KUKA KRL program: MyProgram_149().src

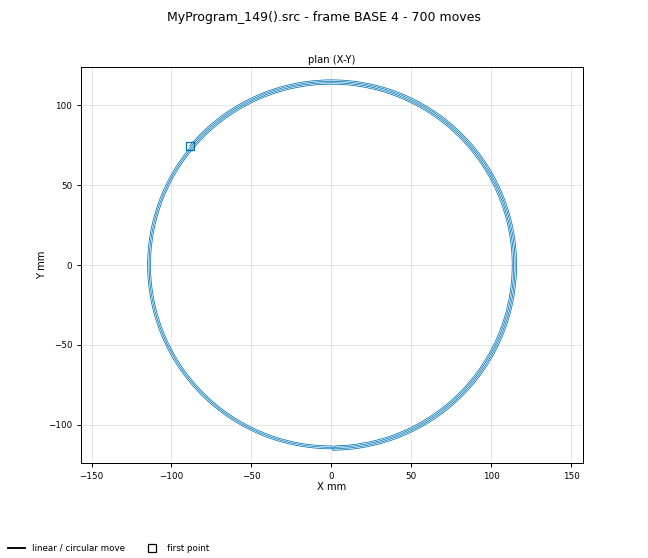
[picture p0: tool path of MyProgram_149().src in frame BASE 4, 700 of 700 moves have a stored position in this frame; points joined in program order, loops and branches not executed]
&ACCESS RVP
&REL 1
&PARAM TEMPLATE = C:\KRC\Roboter\Template\vorgabe
&PARAM EDITMASK = *
DEF MyProgram_149()
; ---- Setting reference (Base) ----
$BASE = BASE_DATA[4]

; --------------------------
; ---- Setting tool (TCP) ----
$TOOL = TOOL_DATA[3]
; --------------------------

$VEL.CP = VEL_APROX_PRINT
Startdeposition()
$VEL.CP = VEL_PRINT
LIN {X -88.6601,Y 74.5291,Z 117,A 135.3963,B 24.9406,C -1.7805,E1 24.8781,E2 310.5914} C_DIS
LIN {X -86.8043,Y 76.6825,Z 117,A 133.9686,B 24.9404,C -1.7832,E1 24.8807,E2 312.019} C_DIS
LIN {X -84.8592,Y 78.8302,Z 117,A 132.5273,B 24.9402,C -1.7865,E1 24.8834,E2 313.4588} C_DIS
LIN {X -82.9372,Y 80.8494,Z 117,A 131.1408,B 24.94,C -1.7896,E1 24.8861,E2 314.8439} C_DIS
LIN {X -80.928,Y 82.8605,Z 117,A 129.7272,B 24.9398,C -1.7928,E1 24.8889,E2 316.256} C_DIS
LIN {X -78.8302,Y 84.8592,Z 117,A 128.2864,B 24.9396,C -1.7958,E1 24.8918,E2 317.6954} C_DIS
LIN {X -77.0268,Y 86.497,Z 117,A 127.0345,B 24.9395,C -1.7968,E1 24.8944,E2 318.9501} C_DIS
LIN {X -74.5714,Y 88.625,Z 117,A 125.4601,B 24.9392,C -1.8017,E1 24.8978,E2 320.5189} C_DIS
LIN {X -72.3739,Y 90.4284,Z 117,A 124.0473,B 24.939,C -1.8045,E1 24.9008,E2 321.9303} C_DIS
LIN {X -70.1764,Y 92.1438,Z 117,A 122.6615,B 24.9388,C -1.8072,E1 24.9039,E2 323.3147} C_DIS
LIN {X -67.9234,Y 93.8167,Z 117,A 121.2662,B 24.9386,C -1.8098,E1 24.907,E2 324.7087} C_DIS
LIN {X -65.5706,Y 95.4762,Z 117,A 119.8357,B 24.9384,C -1.8124,E1 24.9103,E2 326.138} C_DIS
LIN {X -63.2077,Y 97.0566,Z 117,A 118.4237,B 24.9383,C -1.8149,E1 24.9136,E2 327.5486} C_DIS
LIN {X -60.7603,Y 98.6077,Z 117,A 116.9852,B 24.9381,C -1.8174,E1 24.917,E2 328.9857} C_DIS
LIN {X -58.3693,Y 100.0412,Z 117,A 115.6133,B 24.9379,C -1.8202,E1 24.9203,E2 330.3551} C_DIS
LIN {X -55.8486,Y 101.4702,Z 117,A 114.162,B 24.9378,C -1.822,E1 24.9238,E2 331.8064} C_DIS
LIN {X -53.3902,Y 102.7847,Z 117,A 112.7778,B 24.9376,C -1.8241,E1 24.9272,E2 333.1894} C_DIS
LIN {X -50.8516,Y 104.064,Z 117,A 111.3658,B 24.9375,C -1.8262,E1 24.9308,E2 334.6002} C_DIS
LIN {X -48.2327,Y 105.3038,Z 117,A 109.9286,B 24.9373,C -1.8282,E1 24.9344,E2 336.0362} C_DIS
LIN {X -45.6339,Y 106.4558,Z 117,A 108.5177,B 24.9373,C -1.8301,E1 24.938,E2 337.4458} C_DIS
LIN {X -43.0076,Y 107.5436,Z 117,A 107.1073,B 24.9371,C -1.8319,E1 24.9417,E2 338.8551} C_DIS
LIN {X -40.3554,Y 108.5667,Z 117,A 105.697,B 24.937,C -1.8336,E1 24.9453,E2 340.2643} C_DIS
LIN {X -37.6788,Y 109.5243,Z 117,A 104.2869,B 24.9369,C -1.8352,E1 24.949,E2 341.6734} C_DIS
LIN {X -34.9796,Y 110.416,Z 117,A 102.8769,B 24.9368,C -1.8368,E1 24.9528,E2 343.0823} C_DIS
LIN {X -32.312,Y 111.2256,Z 117,A 101.4947,B 24.9367,C -1.8382,E1 24.9565,E2 344.4636} C_DIS
LIN {X -29.5726,Y 111.9851,Z 117,A 100.0842,B 24.9366,C -1.8394,E1 24.9603,E2 345.8732} C_DIS
LIN {X -26.8155,Y 112.6771,Z 117,A 98.6751,B 24.9365,C -1.8407,E1 24.9641,E2 347.2813} C_DIS
LIN {X -24.0422,Y 113.3013,Z 117,A 97.2672,B 24.9365,C -1.8418,E1 24.9679,E2 348.6881} C_DIS
LIN {X -21.5271,Y 113.8047,Z 117,A 95.9717,B 24.9365,C -1.8418,E1 24.9715,E2 349.9852} C_DIS
LIN {X -18.8927,Y 114.2711,Z 117,A 94.6168,B 24.9365,C -1.8414,E1 24.9752,E2 351.3423} C_DIS
LIN {X -15.5877,Y 114.7706,Z 117,A 93.0146,B 24.9362,C -1.8446,E1 24.9796,E2 352.9381} C_DIS
LIN {X -12.8209,Y 115.1122,Z 117,A 91.6457,B 24.9362,C -1.8459,E1 24.9834,E2 354.305} C_DIS
LIN {X -9.9921,Y 115.3922,Z 117,A 90.226,B 24.9362,C -1.8459,E1 24.9874,E2 355.7252} C_DIS
LIN {X -7.1024,Y 115.6064,Z 117,A 88.7913,B 24.9361,C -1.8465,E1 24.9914,E2 357.1591} C_DIS
LIN {X -4.3917,Y 115.7403,Z 117,A 87.4449,B 24.9361,C -1.8468,E1 24.9951,E2 358.5052} C_DIS
LIN {X -1.4213,Y 115.8156,Z 117,A 85.9771,B 24.9361,C -1.8473,E1 24.9992,E2 359.972} C_DIS
LIN {X 1.4213,Y 115.8156,Z 117,A 84.5704,B 24.9361,C -1.8475,E1 25.0032,E2 361.378} C_DIS
LIN {X 4.2632,Y 115.7459,Z 117,A 83.1636,B 24.9361,C -1.8476,E1 25.0071,E2 362.7843} C_DIS
LIN {X 7.0476,Y 115.6094,Z 117,A 81.7846,B 24.9361,C -1.8476,E1 25.0109,E2 364.1626} C_DIS
LIN {X 9.9374,Y 115.3973,Z 117,A 80.3512,B 24.9361,C -1.8476,E1 25.0149,E2 365.5955} C_DIS
LIN {X 12.2215,Y 115.1757,Z 117,A 79.1531,B 24.9362,C -1.8447,E1 25.0183,E2 366.7997} C_DIS
LIN {X 15.5877,Y 114.7706,Z 117,A 77.54,B 24.936,C -1.8471,E1 25.0227,E2 368.4058} C_DIS
LIN {X 17.9447,Y 114.4239,Z 117,A 76.3162,B 24.9362,C -1.8448,E1 25.0261,E2 369.6339} C_DIS
LIN {X 20.7205,Y 113.9539,Z 117,A 74.924,B 24.9362,C -1.8443,E1 25.0299,E2 371.0257} C_DIS
LIN {X 23.9885,Y 113.313,Z 117,A 73.3247,B 24.9362,C -1.8456,E1 25.0343,E2 372.62} C_DIS
LIN {X 26.7087,Y 112.7025,Z 117,A 71.9472,B 24.9362,C -1.845,E1 25.038,E2 373.9971} C_DIS
LIN {X 29.4665,Y 112.0131,Z 117,A 70.5426,B 24.9362,C -1.8442,E1 25.0418,E2 375.4014} C_DIS
LIN {X 32.2594,Y 111.2412,Z 117,A 69.1115,B 24.9363,C -1.8433,E1 25.0457,E2 376.8323} C_DIS
LIN {X 34.9272,Y 110.4323,Z 117,A 67.7347,B 24.9363,C -1.8423,E1 25.0493,E2 378.2089} C_DIS
LIN {X 37.3427,Y 109.6377,Z 117,A 66.4515,B 24.9365,C -1.8401,E1 25.0528,E2 379.4947} C_DIS
LIN {X 40.3038,Y 108.5855,Z 117,A 64.9276,B 24.9365,C -1.8401,E1 25.0567,E2 381.0157} C_DIS
LIN {X 43.0076,Y 107.5436,Z 117,A 63.4973,B 24.9366,C -1.8387,E1 25.0605,E2 382.4459} C_DIS
LIN {X 45.4321,Y 106.5408,Z 117,A 62.1891,B 24.9368,C -1.8369,E1 25.0638,E2 383.7554} C_DIS
LIN {X 47.998,Y 105.4096,Z 117,A 60.8009,B 24.9368,C -1.8353,E1 25.0674,E2 385.144} C_DIS
LIN {X 50.8024,Y 104.0884,Z 117,A 59.2892,B 24.9369,C -1.8343,E1 25.0712,E2 386.654} C_DIS
LIN {X 53.2927,Y 102.8353,Z 117,A 57.9128,B 24.937,C -1.8327,E1 25.0746,E2 388.0306} C_DIS
LIN {X 55.8486,Y 101.4702,Z 117,A 56.4846,B 24.9372,C -1.8309,E1 25.0781,E2 389.4588} C_DIS
LIN {X 58.322,Y 100.0691,Z 117,A 55.0826,B 24.9372,C -1.8291,E1 25.0815,E2 390.8609} C_DIS
LIN {X 60.7133,Y 98.6362,Z 117,A 53.7195,B 24.9374,C -1.8277,E1 25.0848,E2 392.223} C_DIS
LIN {X 63.1157,Y 97.1165,Z 117,A 52.3067,B 24.9376,C -1.8252,E1 25.0881,E2 393.6373} C_DIS
LIN {X 65.1708,Y 95.7477,Z 117,A 51.045,B 24.9378,C -1.8214,E1 25.091,E2 394.9036} C_DIS
LIN {X 67.8497,Y 93.8707,Z 117,A 49.4771,B 24.9378,C -1.8208,E1 25.0946,E2 396.4674} C_DIS
LIN {X 70.089,Y 92.2103,Z 117,A 48.1024,B 24.938,C -1.8186,E1 25.0976,E2 397.8425} C_DIS
LIN {X 72.3739,Y 90.4284,Z 117,A 46.6755,B 24.9382,C -1.8162,E1 25.1008,E2 399.2697} C_DIS
LIN {X 75.2543,Y 88.0431,Z 117,A 44.7753,B 24.9386,C -1.8104,E1 25.1049,E2 401.1763} C_DIS
LIN {X 77.7829,Y 85.8202,Z 117,A 43.1751,B 24.9386,C -1.8099,E1 25.1082,E2 402.7712} C_DIS
LIN {X 79.8656,Y 83.8854,Z 117,A 41.7751,B 24.9388,C -1.8073,E1 25.111,E2 404.1717} C_DIS
LIN {X 81.9002,Y 81.9002,Z 117,A 40.3751,B 24.939,C -1.8046,E1 25.1138,E2 405.5723} C_DIS
LIN {X 83.8854,Y 79.8656,Z 117,A 38.9755,B 24.9392,C -1.8018,E1 25.1165,E2 406.9723} C_DIS
LIN {X 85.7831,Y 77.8233,Z 117,A 37.6053,B 24.9393,C -1.7991,E1 25.1191,E2 408.343} C_DIS
LIN {X 87.3549,Y 76.0521,Z 117,A 36.3734,B 24.9397,C -1.7936,E1 25.1214,E2 409.5821} C_DIS
LIN {X 89.5334,Y 73.4782,Z 117,A 34.778,B 24.9397,C -1.793,E1 25.1242,E2 411.1718} C_DIS
LIN {X 91.3097,Y 71.2588,Z 117,A 33.3787,B 24.94,C -1.7899,E1 25.1267,E2 412.5718} C_DIS
LIN {X 92.7838,Y 69.3256,Z 117,A 32.141,B 24.9403,C -1.7853,E1 25.1288,E2 413.8144} C_DIS
LIN {X 94.6962,Y 66.6926,Z 117,A 30.5813,B 24.9403,C -1.7835,E1 25.1313,E2 415.3707} C_DIS
LIN {X 96.3044,Y 64.3486,Z 117,A 29.1828,B 24.9406,C -1.7803,E1 25.1335,E2 416.77} C_DIS
LIN {X 97.7753,Y 62.0892,Z 117,A 27.8528,B 24.9408,C -1.7769,E1 25.1355,E2 418.1011} C_DIS
LIN {X 99.3459,Y 59.5456,Z 117,A 26.3861,B 24.941,C -1.7735,E1 25.1376,E2 419.5684} C_DIS
LIN {X 100.7561,Y 57.1265,Z 117,A 25.0092,B 24.9413,C -1.7702,E1 25.1395,E2 420.9462} C_DIS
LIN {X 102.1218,Y 54.6475,Z 117,A 23.6172,B 24.9415,C -1.7667,E1 25.1414,E2 422.3391} C_DIS
LIN {X 103.4321,Y 52.1248,Z 117,A 22.2197,B 24.9417,C -1.7631,E1 25.1432,E2 423.7375} C_DIS
LIN {X 104.704,Y 49.5213,Z 117,A 20.7949,B 24.942,C -1.7595,E1 25.1449,E2 425.1633} C_DIS
LIN {X 105.8877,Y 46.9368,Z 117,A 19.3972,B 24.9422,C -1.7558,E1 25.1465,E2 426.5621} C_DIS
LIN {X 107.0077,Y 44.3241,Z 117,A 17.9997,B 24.9425,C -1.7521,E1 25.148,E2 427.9607} C_DIS
LIN {X 108.0633,Y 41.6846,Z 117,A 16.6022,B 24.9427,C -1.7484,E1 25.1495,E2 429.3592} C_DIS
LIN {X 108.9986,Y 39.1713,Z 117,A 15.2768,B 24.943,C -1.7445,E1 25.1507,E2 430.6864} C_DIS
LIN {X 109.9785,Y 36.332,Z 117,A 13.8078,B 24.9432,C -1.7408,E1 25.152,E2 432.1558} C_DIS
LIN {X 110.837,Y 33.622,Z 117,A 12.4107,B 24.9435,C -1.7369,E1 25.1532,E2 433.5541} C_DIS
LIN {X 111.6138,Y 30.9446,Z 117,A 11.0407,B 24.9437,C -1.7331,E1 25.1542,E2 434.9252} C_DIS
LIN {X 112.2551,Y 28.5247,Z 117,A 9.7764,B 24.944,C -1.7281,E1 25.1551,E2 436.194} C_DIS
LIN {X 112.9058,Y 25.8284,Z 117,A 8.3965,B 24.9443,C -1.7234,E1 25.156,E2 437.5769} C_DIS
LIN {X 113.5878,Y 22.65,Z 117,A 6.8501,B 24.9445,C -1.7212,E1 25.1569,E2 439.1195} C_DIS
LIN {X 114.1094,Y 19.8556,Z 117,A 5.4522,B 24.9447,C -1.7172,E1 25.1576,E2 440.5188} C_DIS
LIN {X 114.5623,Y 17.0492,Z 117,A 4.0634,B 24.945,C -1.7135,E1 25.1582,E2 441.9081} C_DIS
LIN {X 114.9462,Y 14.2326,Z 117,A 2.6599,B 24.9453,C -1.7091,E1 25.1587,E2 443.3136} C_DIS
LIN {X 115.2666,Y 11.3528,Z 117,A 1.2365,B 24.9455,C -1.705,E1 25.1591,E2 444.7383} C_DIS
LIN {X 115.5061,Y 8.5753,Z 117,A -0.1344,B 24.9458,C -1.7009,E1 25.1594,E2 446.1106} C_DIS
LIN {X 115.6818,Y 5.738,Z 117,A -1.5297,B 24.946,C -1.6969,E1 25.1596,E2 447.5072} C_DIS
LIN {X 115.7878,Y 2.8973,Z 117,A -2.9272,B 24.9463,C -1.6927,E1 25.1598,E2 448.9062} C_DIS
LIN {X 115.8232,Y 0,Z 117,A -4.3066,B 24.9464,C -1.6906,E1 25.1598,E2 450.2824} C_DIS
LIN {X 115.7905,Y -2.7876,Z 117,A -5.7202,B 24.9468,C -1.6845,E1 25.1598,E2 451.7021} C_DIS
LIN {X 115.6848,Y -5.6832,Z 117,A -7.1426,B 24.9471,C -1.6803,E1 25.1595,E2 453.1257} C_DIS
LIN {X 115.5142,Y -8.4658,Z 117,A -8.5122,B 24.9473,C -1.6763,E1 25.1593,E2 454.4968} C_DIS
LIN {X 115.2666,Y -11.3528,Z 117,A -9.9355,B 24.9476,C -1.6721,E1 25.1589,E2 455.9216} C_DIS
LIN {X 115.0189,Y -13.6181,Z 117,A -11.1264,B 24.948,C -1.6654,E1 25.1585,E2 457.1211} C_DIS
LIN {X 114.5784,Y -16.9406,Z 117,A -12.7024,B 24.9481,C -1.6639,E1 25.1579,E2 458.6915} C_DIS
LIN {X 114.1282,Y -19.7474,Z 117,A -14.0981,B 24.9484,C -1.6598,E1 25.1573,E2 460.0886} C_DIS
LIN {X 113.6092,Y -22.5423,Z 117,A -15.4956,B 24.9486,C -1.6556,E1 25.1566,E2 461.4877} C_DIS
LIN {X 113.0101,Y -25.3773,Z 117,A -16.9181,B 24.9489,C -1.6515,E1 25.1557,E2 462.9116} C_DIS
LIN {X 112.423,Y -27.8569,Z 117,A -18.1889,B 24.9492,C -1.647,E1 25.1549,E2 464.1857} C_DIS
LIN {X 111.6287,Y -30.8918,Z 117,A -19.7114,B 24.9494,C -1.6434,E1 25.1538,E2 465.708} C_DIS
LIN {X 110.837,Y -33.622,Z 117,A -21.108,B 24.9496,C -1.6394,E1 25.1527,E2 467.106} C_DIS
LIN {X 109.9954,Y -36.2798,Z 117,A -22.4779,B 24.9499,C -1.6354,E1 25.1515,E2 468.4775} C_DIS
LIN {X 109.0719,Y -38.9682,Z 117,A -23.8756,B 24.9501,C -1.6314,E1 25.1502,E2 469.8769} C_DIS
LIN {X 108.1211,Y -41.5319,Z 117,A -25.2235,B 24.9504,C -1.6274,E1 25.1489,E2 471.2266} C_DIS
LIN {X 107.0284,Y -44.2732,Z 117,A -26.6685,B 24.9506,C -1.6236,E1 25.1473,E2 472.6727} C_DIS
LIN {X 105.9097,Y -46.8865,Z 117,A -28.0665,B 24.9508,C -1.6196,E1 25.1458,E2 474.0724} C_DIS
LIN {X 104.8874,Y -49.1273,Z 117,A -29.3169,B 24.9512,C -1.6144,E1 25.1443,E2 475.3283} C_DIS
LIN {X 103.4571,Y -52.0759,Z 117,A -30.8867,B 24.9513,C -1.6119,E1 25.1424,E2 476.8956} C_DIS
LIN {X 102.1479,Y -54.5992,Z 117,A -32.2841,B 24.9515,C -1.6081,E1 25.1406,E2 478.2945} C_DIS
LIN {X 100.804,Y -57.0417,Z 117,A -33.6543,B 24.9518,C -1.6045,E1 25.1387,E2 479.6662} C_DIS
LIN {X 99.3738,Y -59.4984,Z 117,A -35.0515,B 24.952,C -1.6008,E1 25.1367,E2 481.0649} C_DIS
LIN {X 97.8837,Y -61.9192,Z 117,A -36.4495,B 24.9522,C -1.5971,E1 25.1346,E2 482.4645} C_DIS
LIN {X 96.3044,Y -64.3486,Z 117,A -37.8741,B 24.9524,C -1.5935,E1 25.1325,E2 483.8907} C_DIS
LIN {X 94.6962,Y -66.6926,Z 117,A -39.2719,B 24.9526,C -1.5899,E1 25.1302,E2 485.29} C_DIS
LIN {X 93.031,Y -68.9965,Z 117,A -40.6701,B 24.9528,C -1.5864,E1 25.1279,E2 486.6897} C_DIS
LIN {X 91.3097,Y -71.2588,Z 117,A -42.0682,B 24.9531,C -1.583,E1 25.1255,E2 488.0893} C_DIS
LIN {X 89.568,Y -73.4355,Z 117,A -43.4392,B 24.9532,C -1.5796,E1 25.1231,E2 489.4617} C_DIS
LIN {X 87.7388,Y -75.6115,Z 117,A -44.8377,B 24.9534,C -1.5763,E1 25.1206,E2 490.8617} C_DIS
LIN {X 85.8202,Y -77.7829,Z 117,A -46.2631,B 24.9536,C -1.573,E1 25.1179,E2 492.2887} C_DIS
LIN {X 83.8854,Y -79.8656,Z 117,A -47.6618,B 24.9538,C -1.5698,E1 25.1153,E2 493.6888} C_DIS
LIN {X 81.9002,Y -81.9002,Z 117,A -49.0605,B 24.954,C -1.5666,E1 25.1125,E2 495.089} C_DIS
LIN {X 79.9051,Y -83.8473,Z 117,A -50.4328,B 24.9542,C -1.5636,E1 25.1097,E2 496.4627} C_DIS
LIN {X 77.9197,Y -85.6946,Z 117,A -51.7743,B 24.9544,C -1.5604,E1 25.107,E2 497.8062} C_DIS
LIN {X 75.8953,Y -87.4919,Z 117,A -53.1262,B 24.9546,C -1.5567,E1 25.1041,E2 499.1615} C_DIS
LIN {X 73.5526,Y -89.4716,Z 117,A -54.6127,B 24.9547,C -1.5547,E1 25.101,E2 500.6471} C_DIS
LIN {X 71.3019,Y -91.2757,Z 117,A -56.03,B 24.9549,C -1.552,E1 25.0978,E2 502.0655} C_DIS
LIN {X 69.0404,Y -92.998,Z 117,A -57.43,B 24.955,C -1.5493,E1 25.0947,E2 503.4669} C_DIS
LIN {X 66.6926,Y -94.6962,Z 117,A -58.8567,B 24.9552,C -1.5466,E1 25.0915,E2 504.8949} C_DIS
LIN {X 64.3486,Y -96.3044,Z 117,A -60.2571,B 24.9553,C -1.544,E1 25.0882,E2 506.2966} C_DIS
LIN {X 61.966,Y -97.8545,Z 117,A -61.6573,B 24.9555,C -1.5416,E1 25.0849,E2 507.6982} C_DIS
LIN {X 59.5456,Y -99.3458,Z 117,A -63.0579,B 24.9556,C -1.5392,E1 25.0816,E2 509.1} C_DIS
LIN {X 57.0896,Y -100.7773,Z 117,A -64.4588,B 24.9557,C -1.5368,E1 25.0782,E2 510.5023} C_DIS
LIN {X 54.6475,Y -102.1218,Z 117,A -65.8328,B 24.9559,C -1.5347,E1 25.0748,E2 511.8774} C_DIS
LIN {X 52.1248,Y -103.4321,Z 117,A -67.2339,B 24.9559,C -1.5325,E1 25.0713,E2 513.2797} C_DIS
LIN {X 49.5213,Y -104.704,Z 117,A -68.6624,B 24.9561,C -1.5304,E1 25.0677,E2 514.7094} C_DIS
LIN {X 47.1001,Y -105.8142,Z 117,A -69.9814,B 24.9562,C -1.5283,E1 25.0644,E2 516.0301} C_DIS
LIN {X 44.3241,Y -107.0077,Z 117,A -71.4657,B 24.9563,C -1.5266,E1 25.0606,E2 517.5151} C_DIS
LIN {X 41.6846,Y -108.0633,Z 117,A -72.8677,B 24.9564,C -1.5248,E1 25.0569,E2 518.9182} C_DIS
LIN {X 39.0716,Y -109.0349,Z 117,A -74.2406,B 24.9565,C -1.5232,E1 25.0533,E2 520.2919} C_DIS
LIN {X 36.7201,Y -109.8476,Z 117,A -75.5113,B 24.9567,C -1.5199,E1 25.0499,E2 521.568} C_DIS
LIN {X 33.622,Y -110.837,Z 117,A -77.0751,B 24.9567,C -1.5199,E1 25.0458,E2 523.1288} C_DIS
LIN {X 30.9446,Y -111.6138,Z 117,A -78.4508,B 24.9567,C -1.5186,E1 25.0421,E2 524.5054} C_DIS
LIN {X 28.143,Y -112.3532,Z 117,A -79.8811,B 24.9569,C -1.5172,E1 25.0382,E2 525.9368} C_DIS
LIN {X 25.3773,Y -113.0101,Z 117,A -81.2845,B 24.9569,C -1.516,E1 25.0344,E2 527.3411} C_DIS
LIN {X 22.65,Y -113.5878,Z 117,A -82.6618,B 24.957,C -1.5149,E1 25.0306,E2 528.7194} C_DIS
LIN {X 19.8015,Y -114.1191,Z 117,A -84.092,B 24.957,C -1.5139,E1 25.0267,E2 530.1504} C_DIS
LIN {X 17.0492,Y -114.5623,Z 117,A -85.4699,B 24.9571,C -1.5129,E1 25.0229,E2 531.5292} C_DIS
LIN {X 14.2326,Y -114.9462,Z 117,A -86.8675,B 24.9571,C -1.5124,E1 25.019,E2 532.927} C_DIS
LIN {X 11.3528,Y -115.2666,Z 117,A -88.3045,B 24.9572,C -1.5114,E1 25.015,E2 534.3654} C_DIS
LIN {X 8.5206,Y -115.5105,Z 117,A -89.7097,B 24.9572,C -1.5107,E1 25.0111,E2 535.7713} C_DIS
LIN {X 5.6832,Y -115.6848,Z 117,A -91.1143,B 24.9572,C -1.5102,E1 25.0072,E2 537.1767} C_DIS
LIN {X 2.8973,Y -115.7878,Z 117,A -92.4935,B 24.9572,C -1.5098,E1 25.0033,E2 538.5567} C_DIS
LIN {X 0.8116,Y -115.8194,Z 117,A -93.2511,B 24.9566,C -1.5217,E1 25.0013,E2 539.2858} C_DIS
Enddeposition()
LIN {X 0.8116,Y -115.8194,Z 117,A -93.2511,B 24.9566,C -1.5217,E1 25.0013,E2 539.2858} C_DIS
Startdeposition()
$VEL.CP = VEL_PRINT
LIN {X 1.2098,Y -114.9149,Z 117,A -92.7013,B 24.9548,C -1.5531,E1 25.0031,E2 538.6618} C_DIS
LIN {X 3.6789,Y -114.8613,Z 117,A -91.2682,B 24.9543,C -1.5625,E1 25.0071,E2 537.2068} C_DIS
LIN {X 7.8843,Y -114.6494,Z 117,A -89.5393,B 24.9552,C -1.5468,E1 25.0118,E2 535.5156} C_DIS
LIN {X 11.3435,Y -114.3604,Z 117,A -87.5384,B 24.9544,C -1.5598,E1 25.0175,E2 533.4852} C_DIS
LIN {X 14.8457,Y -113.9572,Z 117,A -85.8672,B 24.9546,C -1.557,E1 25.0221,E2 531.8217} C_DIS
LIN {X 18.1047,Y -113.4864,Z 117,A -84.1715,B 24.9544,C -1.5606,E1 25.0268,E2 530.1191} C_DIS
LIN {X 20.9728,Y -112.992,Z 117,A -82.8451,B 24.9546,C -1.5562,E1 25.0304,E2 528.8047} C_DIS
LIN {X 25.3486,Y -112.0909,Z 117,A -80.5045,B 24.9542,C -1.5633,E1 25.0368,E2 526.4503} C_DIS
LIN {X 28.3498,Y -111.3687,Z 117,A -79.1593,B 24.9546,C -1.5561,E1 25.0404,E2 525.1241} C_DIS
LIN {X 30.6536,Y -110.7586,Z 117,A -77.8777,B 24.9543,C -1.5616,E1 25.0439,E2 523.8316} C_DIS
LIN {X 32.906,Y -110.1085,Z 117,A -76.5354,B 24.9538,C -1.5708,E1 25.0475,E2 522.4697} C_DIS
LIN {X 36.4786,Y -108.9771,Z 117,A -74.7175,B 24.9538,C -1.5708,E1 25.0524,E2 520.6553} C_DIS
LIN {X 40.4692,Y -107.559,Z 117,A -72.8108,B 24.9542,C -1.5643,E1 25.0573,E2 518.7679} C_DIS
LIN {X 42.6984,Y -106.6956,Z 117,A -71.3945,B 24.9535,C -1.5762,E1 25.0611,E2 517.3266} C_DIS
LIN {X 46.2055,Y -105.2225,Z 117,A -69.6792,B 24.9538,C -1.5708,E1 25.0654,E2 515.6283} C_DIS
LIN {X 49.1533,Y -103.88,Z 117,A -67.8577,B 24.9531,C -1.5828,E1 25.0701,E2 513.783} C_DIS
LIN {X 52.8895,Y -102.0283,Z 117,A -65.8043,B 24.9529,C -1.5851,E1 25.0752,E2 511.7298} C_DIS
LIN {X 56.3625,Y -100.1501,Z 117,A -63.4079,B 24.9515,C -1.6085,E1 25.0812,E2 509.2852} C_DIS
LIN {X 59.9119,Y -98.0677,Z 117,A -61.9666,B 24.953,C -1.584,E1 25.0845,E2 507.9062} C_DIS
LIN {X 61.8888,Y -96.8322,Z 117,A -60.7786,B 24.9528,C -1.5874,E1 25.0873,E2 506.7139} C_DIS
LIN {X 64.1436,Y -95.3538,Z 117,A -59.5511,B 24.9529,C -1.5847,E1 25.0901,E2 505.497} C_DIS
LIN {X 66.0888,Y -94.0174,Z 117,A -57.9839,B 24.9517,C -1.6052,E1 25.0938,E2 503.8867} C_DIS
LIN {X 69.9248,Y -91.1989,Z 117,A -55.8663,B 24.9521,C -1.5984,E1 25.0985,E2 501.7928} C_DIS
LIN {X 72.3813,Y -89.2613,Z 117,A -54.2134,B 24.9517,C -1.6062,E1 25.1021,E2 500.1276} C_DIS
LIN {X 75.2854,Y -86.8269,Z 117,A -52.645,B 24.9523,C -1.5956,E1 25.1053,E2 498.5904} C_DIS
LIN {X 77.4854,Y -84.8689,Z 117,A -50.9734,B 24.9515,C -1.6085,E1 25.1089,E2 496.8951} C_DIS
LIN {X 80.0003,Y -82.5028,Z 117,A -49.3117,B 24.9515,C -1.6099,E1 25.1122,E2 495.237} C_DIS
LIN {X 82.4878,Y -80.0159,Z 117,A -47.5085,B 24.951,C -1.6165,E1 25.1158,E2 493.4259} C_DIS
LIN {X 86.1776,Y -76.0289,Z 117,A -44.7625,B 24.9505,C -1.6252,E1 25.1209,E2 490.6715} C_DIS
LIN {X 88.1306,Y -73.7549,Z 117,A -43.2861,B 24.9503,C -1.6283,E1 25.1236,E2 489.1945} C_DIS
LIN {X 90.0442,Y -71.4053,Z 117,A -41.9968,B 24.9507,C -1.622,E1 25.1258,E2 487.9262} C_DIS
LIN {X 91.4747,Y -69.5663,Z 117,A -40.7691,B 24.9503,C -1.6282,E1 25.1279,E2 486.6896} C_DIS
LIN {X 92.8911,Y -67.6606,Z 117,A -39.5379,B 24.95,C -1.6337,E1 25.13,E2 485.4513} C_DIS
LIN {X 94.7831,Y -64.9865,Z 117,A -37.6998,B 24.9491,C -1.648,E1 25.1329,E2 483.5886} C_DIS
LIN {X 96.9625,Y -61.6857,Z 117,A -35.9075,B 24.9493,C -1.6451,E1 25.1356,E2 481.812} C_DIS
LIN {X 98.8733,Y -58.5723,Z 117,A -34.3784,B 24.9498,C -1.6367,E1 25.1378,E2 480.3107} C_DIS
LIN {X 100.2696,Y -56.1485,Z 117,A -32.9516,B 24.9495,C -1.6423,E1 25.1398,E2 478.878} C_DIS
LIN {X 101.2258,Y -54.4074,Z 117,A -31.4637,B 24.9478,C -1.6687,E1 25.1418,E2 477.3356} C_DIS
LIN {X 103.4745,Y -49.9973,Z 117,A -29.3447,B 24.9484,C -1.6596,E1 25.1444,E2 475.2493} C_DIS
LIN {X 105.0569,Y -46.5842,Z 117,A -27.5157,B 24.9482,C -1.6631,E1 25.1465,E2 473.422} C_DIS
LIN {X 105.9765,Y -44.4484,Z 117,A -26.1858,B 24.9474,C -1.6748,E1 25.148,E2 472.0719} C_DIS
LIN {X 107.2645,Y -41.2469,Z 117,A -24.4408,B 24.947,C -1.6813,E1 25.1498,E2 470.3213} C_DIS
LIN {X 108.3971,Y -38.167,Z 117,A -23.1047,B 24.9476,C -1.6722,E1 25.151,E2 469.014} C_DIS
LIN {X 109.1361,Y -36.0054,Z 117,A -21.9046,B 24.9472,C -1.6787,E1 25.1521,E2 467.8054} C_DIS
LIN {X 110.1267,Y -32.8448,Z 117,A -20.1785,B 24.9466,C -1.6875,E1 25.1535,E2 466.0684} C_DIS
LIN {X 110.935,Y -30.0011,Z 117,A -18.2953,B 24.9451,C -1.7117,E1 25.1549,E2 464.139} C_DIS
LIN {X 111.8375,Y -26.4452,Z 117,A -16.8441,B 24.9459,C -1.6996,E1 25.1558,E2 462.7248} C_DIS
LIN {X 112.5437,Y -23.2504,Z 117,A -15.2997,B 24.9458,C -1.7007,E1 25.1567,E2 461.1866} C_DIS
LIN {X 113.2613,Y -19.4624,Z 117,A -13.1544,B 24.9447,C -1.7176,E1 25.1578,E2 459.0143} C_DIS
LIN {X 113.9297,Y -15.0582,Z 117,A -11.1354,B 24.9449,C -1.7152,E1 25.1586,E2 457.0127} C_DIS
LIN {X 114.3995,Y -10.933,Z 117,A -9.0557,B 24.9444,C -1.7224,E1 25.1592,E2 454.9284} C_DIS
LIN {X 114.6916,Y -7.2602,Z 117,A -7.2779,B 24.9442,C -1.7256,E1 25.1595,E2 453.1535} C_DIS
LIN {X 114.8648,Y -3.5644,Z 117,A -5.4181,B 24.9438,C -1.7323,E1 25.1597,E2 451.2889} C_DIS
LIN {X 114.9209,Y 0.0447,Z 117,A -3.5719,B 24.9432,C -1.7404,E1 25.1597,E2 449.4346} C_DIS
LIN {X 114.8458,Y 4.1853,Z 117,A -1.4924,B 24.9427,C -1.7478,E1 25.1597,E2 447.3501} C_DIS
LIN {X 114.624,Y 8.2601,Z 117,A 0.4468,B 24.9427,C -1.7499,E1 25.1593,E2 445.4175} C_DIS
LIN {X 114.3962,Y 10.9685,Z 117,A 2.3157,B 24.9407,C -1.7787,E1 25.1588,E2 443.4919} C_DIS
LIN {X 113.9176,Y 15.1513,Z 117,A 3.9305,B 24.9418,C -1.7623,E1 25.1582,E2 441.9251} C_DIS
LIN {X 113.3315,Y 19.0424,Z 117,A 5.6967,B 24.942,C -1.7593,E1 25.1574,E2 440.1764} C_DIS
LIN {X 111.8917,Y 26.211,Z 117,A 9.4772,B 24.9408,C -1.7771,E1 25.1553,E2 436.376} C_DIS
LIN {X 110.9136,Y 30.0801,Z 117,A 11.2864,B 24.941,C -1.7747,E1 25.154,E2 434.5827} C_DIS
LIN {X 110.0384,Y 33.1422,Z 117,A 12.9677,B 24.9403,C -1.784,E1 25.1527,E2 432.8893} C_DIS
LIN {X 108.9126,Y 36.6699,Z 117,A 14.6469,B 24.9405,C -1.7817,E1 25.1512,E2 431.2248} C_DIS
LIN {X 108.1143,Y 38.9631,Z 117,A 15.8161,B 24.9404,C -1.7834,E1 25.1501,E2 430.0582} C_DIS
LIN {X 106.9404,Y 42.0761,Z 117,A 17.6294,B 24.9396,C -1.7956,E1 25.1483,E2 428.2263} C_DIS
LIN {X 105.5383,Y 45.4811,Z 117,A 19.3784,B 24.9395,C -1.7969,E1 25.1464,E2 426.484} C_DIS
LIN {X 104.2964,Y 48.2593,Z 117,A 21.1725,B 24.9383,C -1.8142,E1 25.1443,E2 424.6586} C_DIS
LIN {X 102.6069,Y 51.7574,Z 117,A 22.8621,B 24.9387,C -1.8081,E1 25.1422,E2 422.9926} C_DIS
LIN {X 101.1138,Y 54.6139,Z 117,A 24.3154,B 24.9389,C -1.8054,E1 25.1404,E2 421.5532} C_DIS
LIN {X 100.0352,Y 56.5683,Z 117,A 25.755,B 24.9377,C -1.8237,E1 25.1383,E2 420.0781} C_DIS
LIN {X 97.7913,Y 60.3646,Z 117,A 27.689,B 24.9381,C -1.8172,E1 25.1356,E2 418.1691} C_DIS
LIN {X 96.5777,Y 62.2852,Z 117,A 29.1257,B 24.9369,C -1.8344,E1 25.1334,E2 416.6992} C_DIS
LIN {X 94.3098,Y 65.6682,Z 117,A 30.989,B 24.9371,C -1.8318,E1 25.1305,E2 414.8512} C_DIS
LIN {X 92.1315,Y 68.692,Z 117,A 32.6995,B 24.9373,C -1.8296,E1 25.1277,E2 413.154} C_DIS
LIN {X 88.04,Y 73.8639,Z 117,A 36.1641,B 24.9361,C -1.8456,E1 25.1216,E2 409.6677} C_DIS
LIN {X 84.0193,Y 78.4066,Z 117,A 38.8882,B 24.9366,C -1.8387,E1 25.1165,E2 406.9722} C_DIS
LIN {X 81.8636,Y 80.6536,Z 117,A 40.5703,B 24.936,C -1.848,E1 25.1132,E2 405.2752} C_DIS
LIN {X 79.6601,Y 82.8307,Z 117,A 43.3096,B 24.9319,C -1.9066,E1 25.1075,E2 402.4088} C_DIS
LIN {X 74.5872,Y 87.4265,Z 117,A 45.8601,B 24.9342,C -1.8734,E1 25.1022,E2 399.9469} C_DIS
LIN {X 70.5238,Y 90.7373,Z 117,A 48.223,B 24.9347,C -1.8667,E1 25.0971,E2 397.6084} C_DIS
LIN {X 67.3246,Y 93.1371,Z 117,A 50.1355,B 24.9347,C -1.8665,E1 25.0928,E2 395.7033} C_DIS
LIN {X 64.5759,Y 95.0612,Z 117,A 51.86,B 24.9343,C -1.8717,E1 25.0889,E2 393.9723} C_DIS
LIN {X 61.1525,Y 97.2991,Z 117,A 53.6095,B 24.935,C -1.8619,E1 25.0848,E2 392.2519} C_DIS
LIN {X 58.5283,Y 98.8993,Z 117,A 55.1659,B 24.9348,C -1.8653,E1 25.0811,E2 390.6923} C_DIS
LIN {X 56.0201,Y 100.3413,Z 117,A 56.7599,B 24.9342,C -1.8742,E1 25.0772,E2 389.0821} C_DIS
LIN {X 53.1749,Y 101.8786,Z 117,A 58.2881,B 24.9342,C -1.8725,E1 25.0734,E2 387.562} C_DIS
LIN {X 46.1341,Y 105.2536,Z 117,A 62.1275,B 24.9342,C -1.8748,E1 25.0638,E2 383.7272} C_DIS
LIN {X 42.9658,Y 106.5867,Z 117,A 64.1238,B 24.9331,C -1.8892,E1 25.0585,E2 381.7014} C_DIS
LIN {X 39.5139,Y 107.9134,Z 117,A 65.8727,B 24.9333,C -1.8867,E1 25.054,E2 379.9621} C_DIS
LIN {X 35.6771,Y 109.2423,Z 117,A 67.8133,B 24.9334,C -1.8847,E1 25.0489,E2 378.03} C_DIS
LIN {X 32.0211,Y 110.371,Z 117,A 69.8116,B 24.933,C -1.8901,E1 25.0435,E2 376.0224} C_DIS
LIN {X 28.805,Y 111.2517,Z 117,A 71.472,B 24.933,C -1.8911,E1 25.039,E2 374.3623} C_DIS
LIN {X 24.1663,Y 112.3509,Z 117,A 73.7292,B 24.9332,C -1.8871,E1 25.0329,E2 372.1177} C_DIS
LIN {X 19.824,Y 113.1986,Z 117,A 76.1268,B 24.9326,C -1.8964,E1 25.0263,E2 369.7007} C_DIS
LIN {X 17.0102,Y 113.6556,Z 117,A 77.9714,B 24.9312,C -1.9155,E1 25.0211,E2 367.8128} C_DIS
LIN {X 12.9971,Y 114.1834,Z 117,A 79.3582,B 24.9332,C -1.8881,E1 25.0174,E2 366.4917} C_DIS
LIN {X 8.8009,Y 114.5832,Z 117,A 81.5091,B 24.933,C -1.8905,E1 25.0114,E2 364.3365} C_DIS
LIN {X 5.1762,Y 114.8037,Z 117,A 83.6805,B 24.9319,C -1.9061,E1 25.0053,E2 362.1287} C_DIS
LIN {X -0.609,Y 114.9185,Z 117,A 86.365,B 24.9325,C -1.8969,E1 24.9978,E2 359.4663} C_DIS
LIN {X -4.9468,Y 114.8136,Z 117,A 88.2754,B 24.9334,C -1.8854,E1 24.9926,E2 357.583} C_DIS
LIN {X -11.0074,Y 114.3926,Z 117,A 91.3713,B 24.9333,C -1.8868,E1 24.9839,E2 354.4823} C_DIS
LIN {X -16.4611,Y 113.7355,Z 117,A 94.3856,B 24.9325,C -1.897,E1 24.9755,E2 351.4418} C_DIS
LIN {X -23.3014,Y 112.5332,Z 117,A 97.7356,B 24.9331,C -1.8894,E1 24.9664,E2 348.1063} C_DIS
LIN {X -27.1679,Y 111.6626,Z 117,A 99.6627,B 24.9334,C -1.8855,E1 24.9611,E2 346.1859} C_DIS
LIN {X -29.8429,Y 110.9777,Z 117,A 101.151,B 24.9331,C -1.8888,E1 24.9571,E2 344.6874} C_DIS
LIN {X -33.1987,Y 110.0217,Z 117,A 102.8773,B 24.9333,C -1.8863,E1 24.9525,E2 342.9643} C_DIS
LIN {X -36.0859,Y 109.1095,Z 117,A 104.3798,B 24.9335,C -1.8841,E1 24.9485,E2 341.4641} C_DIS
LIN {X -38.9619,Y 108.1148,Z 117,A 105.8393,B 24.9338,C -1.8798,E1 24.9447,E2 340.012} C_DIS
LIN {X -42.4698,Y 106.7857,Z 117,A 107.5593,B 24.9344,C -1.8709,E1 24.9402,E2 338.3094} C_DIS
LIN {X -45.8461,Y 105.3792,Z 117,A 109.3994,B 24.9345,C -1.869,E1 24.9355,E2 336.4697} C_DIS
LIN {X -48.1855,Y 104.3308,Z 117,A 110.7297,B 24.9345,C -1.8692,E1 24.9321,E2 335.1356} C_DIS
LIN {X -52.8127,Y 102.0675,Z 117,A 114.0614,B 24.9325,C -1.8971,E1 24.9236,E2 331.7288} C_DIS
LIN {X -56.9846,Y 99.7973,Z 117,A 115.7506,B 24.9348,C -1.8644,E1 24.9197,E2 330.1122} C_DIS
LIN {X -60.6889,Y 97.5886,Z 117,A 117.6465,B 24.9359,C -1.8499,E1 24.9152,E2 328.2451} C_DIS
LIN {X -63.2677,Y 95.9366,Z 117,A 119.4564,B 24.9352,C -1.8587,E1 24.9109,E2 326.4085} C_DIS
LIN {X -66.5422,Y 93.6954,Z 117,A 121.1598,B 24.9363,C -1.8433,E1 24.9071,E2 324.7358} C_DIS
LIN {X -68.866,Y 92.0008,Z 117,A 122.7258,B 24.9361,C -1.8458,E1 24.9035,E2 323.1584} C_DIS
LIN {X -71.8267,Y 89.7108,Z 117,A 124.672,B 24.9361,C -1.845,E1 24.8993,E2 321.2069} C_DIS
LIN {X -74.5606,Y 87.4492,Z 117,A 126.5696,B 24.9361,C -1.8464,E1 24.8952,E2 319.2987} C_DIS
LIN {X -77.7773,Y 84.601,Z 117,A 128.7402,B 24.9364,C -1.8426,E1 24.8907,E2 317.1285} C_DIS
LIN {X -80.3588,Y 82.1548,Z 117,A 130.4178,B 24.9369,C -1.8344,E1 24.8873,E2 315.4635} C_DIS
LIN {X -82.1903,Y 80.3229,Z 117,A 131.878,B 24.9367,C -1.8381,E1 24.8844,E2 313.9882} C_DIS
LIN {X -85.0516,Y 77.2863,Z 117,A 133.9655,B 24.937,C -1.8331,E1 24.8805,E2 311.9032} C_DIS
LIN {X -87.1459,Y 74.9166,Z 117,A 135.4008,B 24.9377,C -1.8233,E1 24.8779,E2 310.4849} C_DIS
LIN {X -89.7971,Y 71.7179,Z 117,A 137.571,B 24.9377,C -1.8218,E1 24.8741,E2 308.308} C_DIS
LIN {X -92.26,Y 68.5209,Z 117,A 139.4837,B 24.9384,C -1.8123,E1 24.8708,E2 306.4088} C_DIS
LIN {X -94.1347,Y 65.9201,Z 117,A 141.2197,B 24.9384,C -1.8135,E1 24.868,E2 304.6615} C_DIS
LIN {X -95.6699,Y 63.6722,Z 117,A 143.0397,B 24.9373,C -1.8286,E1 24.8652,E2 302.7966} C_DIS
LIN {X -97.8841,Y 60.214,Z 117,A 144.6181,B 24.939,C -1.8036,E1 24.8629,E2 301.2697} C_DIS
LIN {X -99.9434,Y 56.7303,Z 117,A 146.7418,B 24.9391,C -1.802,E1 24.8599,E2 299.1387} C_DIS
LIN {X -101.7013,Y 53.5115,Z 117,A 148.4792,B 24.9397,C -1.7929,E1 24.8577,E2 297.4138} C_DIS
LIN {X -103.2186,Y 50.5261,Z 117,A 150.2626,B 24.9397,C -1.7925,E1 24.8554,E2 295.6218} C_DIS
LIN {X -105.3423,Y 45.9307,Z 117,A 152.8863,B 24.94,C -1.7889,E1 24.8524,E2 292.9923} C_DIS
LIN {X -107.0883,Y 41.6996,Z 117,A 154.7958,B 24.9415,C -1.7668,E1 24.8505,E2 291.1249} C_DIS
LIN {X -108.4159,Y 38.1134,Z 117,A 156.8745,B 24.9415,C -1.7677,E1 24.8485,E2 289.032} C_DIS
LIN {X -109.3777,Y 35.2586,Z 117,A 158.2675,B 24.942,C -1.7586,E1 24.8473,E2 287.6529} C_DIS
LIN {X -110.0718,Y 33.0297,Z 117,A 159.5635,B 24.942,C -1.7602,E1 24.8462,E2 286.3455} C_DIS
LIN {X -111.0529,Y 29.5646,Z 117,A 161.2652,B 24.9426,C -1.7507,E1 24.845,E2 284.6566} C_DIS
LIN {X -111.6296,Y 27.3032,Z 117,A 162.4051,B 24.9429,C -1.7461,E1 24.8442,E2 283.5211} C_DIS
LIN {X -112.3368,Y 24.2312,Z 117,A 164.1946,B 24.9426,C -1.7498,E1 24.8431,E2 281.7123} C_DIS
LIN {X -113.0969,Y 20.3896,Z 117,A 165.9097,B 24.9437,C -1.7339,E1 24.8422,E2 280.0248} C_DIS
LIN {X -113.523,Y 17.8679,Z 117,A 167.2351,B 24.9437,C -1.7318,E1 24.8416,E2 278.6966} C_DIS
LIN {X -113.9003,Y 15.2852,Z 117,A 168.5271,B 24.9441,C -1.7272,E1 24.8411,E2 277.4079} C_DIS
LIN {X -114.1881,Y 12.9572,Z 117,A 169.9757,B 24.9436,C -1.7346,E1 24.8406,E2 275.9329} C_DIS
LIN {X -114.5756,Y 8.8964,Z 117,A 171.9711,B 24.9441,C -1.7265,E1 24.8402,E2 273.945} C_DIS
LIN {X -114.743,Y 6.3783,Z 117,A 173.6692,B 24.9432,C -1.7402,E1 24.8399,E2 272.2039} C_DIS
LIN {X -114.8944,Y 2.4552,Z 117,A 175.5738,B 24.9438,C -1.7317,E1 24.8398,E2 270.3082} C_DIS
LIN {X -114.915,Y -1.1737,Z 117,A 177.0643,B 24.945,C -1.7129,E1 24.8398,E2 268.8535} C_DIS
LIN {X -114.6943,Y -7.2201,Z 117,A -179.939,B 24.9457,C -1.7023,E1 24.8402,E2 265.864} C_DIS
LIN {X -114.395,Y -10.9812,Z 117,A -177.9865,B 24.9459,C -1.6991,E1 24.8407,E2 263.9074} C_DIS
LIN {X -113.9345,Y -15.0207,Z 117,A -176.0827,B 24.9466,C -1.6877,E1 24.8413,E2 262.0195} C_DIS
LIN {X -113.4172,Y -18.5297,Z 117,A -174.33,B 24.947,C -1.6814,E1 24.8421,E2 260.2713} C_DIS
LIN {X -112.9511,Y -21.1895,Z 117,A -173.0491,B 24.9475,C -1.6745,E1 24.8427,E2 258.9993} C_DIS
LIN {X -112.354,Y -24.1525,Z 117,A -171.4018,B 24.9474,C -1.6755,E1 24.8437,E2 257.3399} C_DIS
LIN {X -111.5882,Y -27.4732,Z 117,A -169.7571,B 24.9479,C -1.668,E1 24.8447,E2 255.7034} C_DIS
LIN {X -110.6996,Y -30.862,Z 117,A -168.1069,B 24.9484,C -1.6587,E1 24.8459,E2 254.0658} C_DIS
LIN {X -109.8732,Y -33.6845,Z 117,A -166.3692,B 24.948,C -1.6652,E1 24.8473,E2 252.3024} C_DIS
LIN {X -108.6518,Y -37.4413,Z 117,A -164.4073,B 24.9484,C -1.659,E1 24.8491,E2 250.3443} C_DIS
LIN {X -107.7191,Y -40.0465,Z 117,A -162.8991,B 24.9484,C -1.6601,E1 24.8505,E2 248.825} C_DIS
LIN {X -106.1046,Y -44.1444,Z 117,A -160.7783,B 24.9489,C -1.6506,E1 24.8527,E2 246.7149} C_DIS
LIN {X -104.5058,Y -47.808,Z 117,A -158.9214,B 24.9496,C -1.6393,E1 24.8548,E2 244.8747} C_DIS
LIN {X -103.2356,Y -50.4918,Z 117,A -157.4744,B 24.95,C -1.6337,E1 24.8566,E2 243.4331} C_DIS
LIN {X -101.1899,Y -54.4736,Z 117,A -155.1012,B 24.95,C -1.6333,E1 24.8597,E2 241.0482} C_DIS
LIN {X -99.4873,Y -57.524,Z 117,A -153.4279,B 24.9505,C -1.6258,E1 24.862,E2 239.3841} C_DIS
LIN {X -97.8185,Y -60.3209,Z 117,A -151.5773,B 24.9502,C -1.6308,E1 24.8647,E2 237.5122} C_DIS
LIN {X -95.3629,Y -64.1302,Z 117,A -149.5306,B 24.9511,C -1.6162,E1 24.8678,E2 235.49} C_DIS
LIN {X -93.7206,Y -66.507,Z 117,A -148.2907,B 24.9518,C -1.6043,E1 24.8697,E2 234.2723} C_DIS
LIN {X -91.8811,Y -69.0253,Z 117,A -146.3976,B 24.9512,C -1.6144,E1 24.8729,E2 232.3461} C_DIS
LIN {X -89.2709,Y -72.3695,Z 117,A -144.3691,B 24.9517,C -1.6057,E1 24.8764,E2 230.3288} C_DIS
LIN {X -87.5141,Y -74.4843,Z 117,A -142.7239,B 24.9512,C -1.6139,E1 24.8795,E2 228.6565} C_DIS
LIN {X -84.5678,Y -77.8136,Z 117,A -140.7222,B 24.952,C -1.5999,E1 24.8832,E2 226.6792} C_DIS
LIN {X -82.0037,Y -80.5118,Z 117,A -138.9083,B 24.9524,C -1.5941,E1 24.8867,E2 224.8713} C_DIS
LIN {X -79.7602,Y -82.7342,Z 117,A -136.9129,B 24.9515,C -1.6085,E1 24.8908,E2 222.8334} C_DIS
LIN {X -77.1781,Y -85.1508,Z 117,A -135.4065,B 24.9524,C -1.594,E1 24.8938,E2 221.3553} C_DIS
LIN {X -75.0537,Y -87.0289,Z 117,A -133.9446,B 24.9524,C -1.5933,E1 24.8969,E2 219.8894} C_DIS
LIN {X -72.2242,Y -89.3886,Z 117,A -132.1871,B 24.9528,C -1.5865,E1 24.9007,E2 218.1413} C_DIS
LIN {X -69.5867,Y -91.4594,Z 117,A -130.6496,B 24.9534,C -1.5778,E1 24.904,E2 216.619} C_DIS
LIN {X -67.54,Y -92.9794,Z 117,A -129.2129,B 24.9531,C -1.5826,E1 24.9073,E2 215.1658} C_DIS
LIN {X -64.3513,Y -95.2132,Z 117,A -127.3528,B 24.9535,C -1.576,E1 24.9116,E2 213.3152} C_DIS
LIN {X -61.2228,Y -97.2552,Z 117,A -125.412,B 24.9535,C -1.5764,E1 24.9162,E2 211.3672} C_DIS
LIN {X -57.6753,Y -99.4004,Z 117,A -123.2959,B 24.9535,C -1.5754,E1 24.9212,E2 209.2469} C_DIS
LIN {X -55.0187,Y -100.8942,Z 117,A -120.6717,B 24.9508,C -1.6211,E1 24.928,E2 206.5068} C_DIS
LIN {X -48.6845,Y -104.0985,Z 117,A -118.5402,B 24.9546,C -1.5559,E1 24.933,E2 204.5248} C_DIS
LIN {X -45.6186,Y -105.4784,Z 117,A -116.5634,B 24.954,C -1.5669,E1 24.9381,E2 202.517} C_DIS
LIN {X -42.4773,Y -106.7828,Z 117,A -114.8462,B 24.954,C -1.5661,E1 24.9426,E2 200.7979} C_DIS
LIN {X -38.4399,Y -108.3013,Z 117,A -112.8533,B 24.9546,C -1.5574,E1 24.9477,E2 198.8218} C_DIS
LIN {X -35.8959,Y -109.1715,Z 117,A -111.605,B 24.9549,C -1.5523,E1 24.951,E2 197.5831} C_DIS
LIN {X -33.3131,Y -109.9877,Z 117,A -110.0108,B 24.9543,C -1.5619,E1 24.9553,E2 195.9635} C_DIS
LIN {X -29.8418,Y -110.978,Z 117,A -107.8964,B 24.9536,C -1.5745,E1 24.9611,E2 193.8159} C_DIS
LIN {X -26.3499,Y -111.8596,Z 117,A -106.0098,B 24.9534,C -1.5776,E1 24.9663,E2 191.9196} C_DIS
LIN {X -22.4595,Y -112.706,Z 117,A -104.4496,B 24.9545,C -1.558,E1 24.9704,E2 190.4038} C_DIS
LIN {X -19.1213,Y -113.3183,Z 117,A -102.8129,B 24.9547,C -1.5551,E1 24.9749,E2 188.7725} C_DIS
LIN {X -15.2422,Y -113.9058,Z 117,A -101.044,B 24.9552,C -1.5464,E1 24.9798,E2 187.0228} C_DIS
LIN {X -12.3684,Y -114.2533,Z 117,A -99.6337,B 24.9552,C -1.5447,E1 24.9837,E2 185.6155} C_DIS
LIN {X -9.4432,Y -114.5318,Z 117,A -97.9964,B 24.9549,C -1.5522,E1 24.9883,E2 183.9597} C_DIS
LIN {X -5.7245,Y -114.7784,Z 117,A -96.0063,B 24.9545,C -1.5581,E1 24.9938,E2 181.9549} C_DIS
LIN {X -2.6939,Y -114.89,Z 117,A -94.5,B 24.9545,C -1.5581,E1 24.9981,E2 180.4485} C_DIS
LIN {X 0.8102,Y -114.9155,Z 117,A -93.5224,B 24.9565,C -1.5245,E1 25.0006,E2 179.5505} C_DIS
Enddeposition()
LIN {X 0.8102,Y -114.9155,Z 117,A -93.5224,B 24.9565,C -1.5245,E1 25.0006,E2 179.5505} C_DIS
Startdeposition()
$VEL.CP = VEL_PRINT
LIN {X 0.143,Y -114.0194,Z 117,A -94.6187,B 24.9574,C -1.5074,E1 24.9974,E2 180.6874} C_DIS
LIN {X -4.3248,Y -113.9375,Z 117,A -96.7021,B 24.9571,C -1.5141,E1 24.9916,E2 182.7553} C_DIS
LIN {X -8.0159,Y -113.7364,Z 117,A -97.7029,B 24.9549,C -1.551,E1 24.9891,E2 183.6689} C_DIS
LIN {X -10.5651,Y -113.5276,Z 117,A -99.9428,B 24.9573,C -1.51,E1 24.9826,E2 186.0072} C_DIS
LIN {X -14.7222,Y -113.0636,Z 117,A -102.1625,B 24.9575,C -1.5054,E1 24.9764,E2 188.2393} C_DIS
LIN {X -19.4528,Y -112.3483,Z 117,A -104.0082,B 24.9562,C -1.5298,E1 24.9715,E2 190.0289} C_DIS
LIN {X -24.6234,Y -111.328,Z 117,A -106.6319,B 24.956,C -1.532,E1 24.9643,E2 192.6504} C_DIS
LIN {X -29.0567,Y -110.2557,Z 117,A -108.9628,B 24.956,C -1.5317,E1 24.958,E2 194.9855} C_DIS
LIN {X -32.6537,Y -109.2425,Z 117,A -110.7436,B 24.9557,C -1.5371,E1 24.9532,E2 196.7563} C_DIS
LIN {X -36.4702,Y -108.028,Z 117,A -112.6835,B 24.9555,C -1.5418,E1 24.9481,E2 198.6886} C_DIS
LIN {X -39.7676,Y -106.8602,Z 117,A -114.7115,B 24.956,C -1.532,E1 24.9427,E2 200.7441} C_DIS
LIN {X -43.6727,Y -105.3245,Z 117,A -116.7752,B 24.9558,C -1.536,E1 24.9374,E2 202.8029} C_DIS
LIN {X -46.8531,Y -103.9467,Z 117,A -118.3532,B 24.9553,C -1.5448,E1 24.9334,E2 204.3637} C_DIS
LIN {X -50.8958,Y -102.0282,Z 117,A -121.0612,B 24.9562,C -1.5284,E1 24.9265,E2 207.1176} C_DIS
LIN {X -54.1887,Y -100.3182,Z 117,A -122.3928,B 24.9548,C -1.553,E1 24.9233,E2 208.3945} C_DIS
LIN {X -57.0285,Y -98.7316,Z 117,A -124.0743,B 24.9548,C -1.5533,E1 24.9192,E2 210.0802} C_DIS
LIN {X -61.6904,Y -95.8876,Z 117,A -126.6183,B 24.9541,C -1.5658,E1 24.9133,E2 212.6025} C_DIS
LIN {X -63.8345,Y -94.4737,Z 117,A -128.7074,B 24.9559,C -1.535,E1 24.9082,E2 214.7718} C_DIS
LIN {X -67.1861,Y -92.1206,Z 117,A -129.9342,B 24.9537,C -1.5726,E1 24.9056,E2 215.9133} C_DIS
LIN {X -70.2461,Y -89.8106,Z 117,A -132.2687,B 24.9544,C -1.5593,E1 24.9004,E2 218.288} C_DIS
LIN {X -72.9661,Y -87.6133,Z 117,A -133.9314,B 24.954,C -1.5665,E1 24.8968,E2 219.9399} C_DIS
LIN {X -75.9939,Y -85.0003,Z 117,A -135.9203,B 24.9537,C -1.5713,E1 24.8926,E2 221.9252} C_DIS
LIN {X -82.0359,Y -79.1848,Z 117,A -139.8257,B 24.9525,C -1.5927,E1 24.8849,E2 225.7959} C_DIS
LIN {X -86.3673,Y -74.4395,Z 117,A -143.3313,B 24.9527,C -1.5886,E1 24.8783,E2 229.3268} C_DIS
LIN {X -89.0682,Y -71.1854,Z 117,A -145.6857,B 24.953,C -1.5844,E1 24.874,E2 231.7022} C_DIS
LIN {X -91.269,Y -68.3383,Z 117,A -147.3154,B 24.9523,C -1.5961,E1 24.8713,E2 233.3119} C_DIS
LIN {X -93.2456,Y -65.6187,Z 117,A -149.2077,B 24.9525,C -1.5921,E1 24.8682,E2 235.2228} C_DIS
LIN {X -95.5222,Y -62.2574,Z 117,A -151.7005,B 24.9533,C -1.5794,E1 24.8643,E2 237.7585} C_DIS
LIN {X -97.7522,Y -58.6941,Z 117,A -153.324,B 24.9518,C -1.6044,E1 24.862,E2 239.3306} C_DIS
LIN {X -101.7983,Y -51.3574,Z 117,A -157.3787,B 24.9507,C -1.6222,E1 24.8567,E2 243.3644} C_DIS
LIN {X -103.028,Y -48.8436,Z 117,A -159.0407,B 24.9511,C -1.616,E1 24.8546,E2 245.0502} C_DIS
LIN {X -104.7591,Y -45.0114,Z 117,A -161.0124,B 24.9504,C -1.6277,E1 24.8524,E2 247.0049} C_DIS
LIN {X -106.1097,Y -41.7236,Z 117,A -163.148,B 24.9509,C -1.6191,E1 24.8502,E2 249.1729} C_DIS
LIN {X -107.5087,Y -37.9744,Z 117,A -164.8427,B 24.9497,C -1.6376,E1 24.8486,E2 250.8331} C_DIS
LIN {X -109.0417,Y -33.3205,Z 117,A -167.1949,B 24.949,C -1.6494,E1 24.8466,E2 253.1707} C_DIS
LIN {X -109.7855,Y -30.7793,Z 117,A -168.6189,B 24.949,C -1.6498,E1 24.8455,E2 254.602} C_DIS
LIN {X -110.7273,Y -27.196,Z 117,A -170.548,B 24.9488,C -1.6529,E1 24.8442,E2 256.5349} C_DIS
LIN {X -111.4193,Y -24.2046,Z 117,A -172.0387,B 24.9484,C -1.6598,E1 24.8433,E2 258.018} C_DIS
LIN {X -112.0346,Y -21.1785,Z 117,A -173.7552,B 24.9484,C -1.6582,E1 24.8423,E2 259.7485} C_DIS
LIN {X -112.6599,Y -17.5467,Z 117,A -175.5336,B 24.9479,C -1.6669,E1 24.8415,E2 261.5166} C_DIS
LIN {X -113.0984,Y -14.4536,Z 117,A -177.0804,B 24.9476,C -1.6728,E1 24.841,E2 263.0585} C_DIS
LIN {X -113.5235,Y -10.6096,Z 117,A -179.0701,B 24.9473,C -1.6773,E1 24.8404,E2 265.0496} C_DIS
LIN {X -113.7823,Y -7.3378,Z 117,A 179.2064,B 24.9471,C -1.6796,E1 24.84,E2 266.7778} C_DIS
LIN {X -113.9741,Y -3.1834,Z 117,A 177.2094,B 24.9465,C -1.6901,E1 24.8398,E2 268.762} C_DIS
LIN {X -114.0055,Y 1.6952,Z 117,A 174.2088,B 24.9473,C -1.6766,E1 24.8398,E2 271.8127} C_DIS
LIN {X -113.8796,Y 5.6541,Z 117,A 172.5788,B 24.946,C -1.6971,E1 24.8401,E2 273.4037} C_DIS
LIN {X -113.645,Y 9.2176,Z 117,A 170.9239,B 24.9453,C -1.7084,E1 24.8404,E2 275.0416} C_DIS
LIN {X -113.3059,Y 12.7351,Z 117,A 169.0065,B 24.9453,C -1.7086,E1 24.841,E2 276.9699} C_DIS
LIN {X -112.8402,Y 16.3494,Z 117,A 167.3173,B 24.9445,C -1.7201,E1 24.8416,E2 278.6417} C_DIS
LIN {X -112.3485,Y 19.452,Z 117,A 165.5724,B 24.9446,C -1.7187,E1 24.8424,E2 280.4004} C_DIS
LIN {X -111.6412,Y 23.1606,Z 117,A 163.7913,B 24.9439,C -1.7294,E1 24.8434,E2 282.1666} C_DIS
LIN {X -110.7896,Y 26.9405,Z 117,A 161.7748,B 24.9437,C -1.7329,E1 24.8446,E2 284.1864} C_DIS
LIN {X -109.8324,Y 30.614,Z 117,A 159.8047,B 24.9435,C -1.7366,E1 24.8461,E2 286.1594} C_DIS
LIN {X -108.7583,Y 34.2345,Z 117,A 158.0748,B 24.9427,C -1.7492,E1 24.8475,E2 287.8692} C_DIS
LIN {X -107.7781,Y 37.2068,Z 117,A 156.2072,B 24.9431,C -1.7425,E1 24.8492,E2 289.7633} C_DIS
LIN {X -106.5731,Y 40.5255,Z 117,A 154.6238,B 24.9422,C -1.7555,E1 24.8507,E2 291.3245} C_DIS
LIN {X -104.9758,Y 44.5001,Z 117,A 152.4591,B 24.9418,C -1.7617,E1 24.853,E2 293.4866} C_DIS
LIN {X -102.3731,Y 50.2006,Z 117,A 149.4275,B 24.9409,C -1.7758,E1 24.8565,E2 296.501} C_DIS
LIN {X -100.7574,Y 53.3679,Z 117,A 147.4246,B 24.9411,C -1.7726,E1 24.8591,E2 298.5222} C_DIS
LIN {X -98.9081,Y 56.7214,Z 117,A 145.5224,B 24.9407,C -1.7792,E1 24.8617,E2 300.4189} C_DIS
LIN {X -96.9754,Y 59.9681,Z 117,A 143.3085,B 24.9411,C -1.7722,E1 24.8649,E2 302.6607} C_DIS
LIN {X -94.2533,Y 64.1601,Z 117,A 140.6212,B 24.9411,C -1.7724,E1 24.8691,E2 305.3611} C_DIS
LIN {X -92.1091,Y 67.2018,Z 117,A 139.2173,B 24.9395,C -1.7959,E1 24.8714,E2 306.7158} C_DIS
LIN {X -87.6603,Y 72.9096,Z 117,A 135.2361,B 24.9398,C -1.792,E1 24.8783,E2 310.7251} C_DIS
LIN {X -84.7514,Y 76.272,Z 117,A 133.2464,B 24.9388,C -1.8074,E1 24.882,E2 312.687} C_DIS
LIN {X -81.952,Y 79.2719,Z 117,A 130.9376,B 24.9391,C -1.8027,E1 24.8864,E2 315.0169} C_DIS
LIN {X -77.8164,Y 83.3361,Z 117,A 128.4855,B 24.9374,C -1.8281,E1 24.8913,E2 317.4187} C_DIS
LIN {X -75.7993,Y 85.1746,Z 117,A 126.964,B 24.9376,C -1.8253,E1 24.8944,E2 318.953} C_DIS
LIN {X -73.4089,Y 87.2442,Z 117,A 125.0941,B 24.9381,C -1.8176,E1 24.8985,E2 320.8485} C_DIS
LIN {X -68.3658,Y 91.2483,Z 117,A 122.0519,B 24.9371,C -1.8323,E1 24.9051,E2 323.8667} C_DIS
LIN {X -65.0976,Y 93.6078,Z 117,A 120.0373,B 24.9368,C -1.8369,E1 24.9097,E2 325.8774} C_DIS
LIN {X -61.8712,Y 95.7715,Z 117,A 117.6125,B 24.9378,C -1.8217,E1 24.9155,E2 328.3463} C_DIS
LIN {X -58.6255,Y 97.7939,Z 117,A 116.2213,B 24.9361,C -1.8466,E1 24.9187,E2 329.6825} C_DIS
LIN {X -56.2183,Y 99.1972,Z 117,A 114.4155,B 24.937,C -1.8327,E1 24.9231,E2 331.5268} C_DIS
LIN {X -51.2106,Y 101.8722,Z 117,A 111.7274,B 24.9363,C -1.8441,E1 24.9297,E2 334.195} C_DIS
LIN {X -47.4779,Y 103.6651,Z 117,A 109.684,B 24.9359,C -1.8489,E1 24.9349,E2 336.2322} C_DIS
LIN {X -41.0644,Y 106.3683,Z 117,A 106.1567,B 24.9357,C -1.8526,E1 24.944,E2 339.7586} C_DIS
LIN {X -37.2159,Y 107.7749,Z 117,A 104.2172,B 24.9351,C -1.8601,E1 24.9491,E2 341.684} C_DIS
LIN {X -33.1588,Y 109.0912,Z 117,A 101.7569,B 24.9359,C -1.8496,E1 24.9557,E2 344.1736} C_DIS
LIN {X -29.1248,Y 110.2373,Z 117,A 99.8201,B 24.9352,C -1.8588,E1 24.9609,E2 346.0916} C_DIS
LIN {X -25.4147,Y 111.1498,Z 117,A 98.0889,B 24.9346,C -1.8685,E1 24.9655,E2 347.8023} C_DIS
LIN {X -21.5737,Y 111.9585,Z 117,A 96.0734,B 24.9346,C -1.8683,E1 24.971,E2 349.8204} C_DIS
LIN {X -18.116,Y 112.5718,Z 117,A 93.3978,B 24.9371,C -1.8319,E1 24.9787,E2 352.5849} C_DIS
LIN {X -12.5703,Y 113.3252,Z 117,A 90.5029,B 24.9372,C -1.83,E1 24.9867,E2 355.486} C_DIS
LIN {X -6.7038,Y 113.8216,Z 117,A 88.7121,B 24.9337,C -1.8799,E1 24.9914,E2 357.1591} C_DIS
LIN {X -0.1698,Y 114.0192,Z 117,A 85.3288,B 24.934,C -1.8766,E1 25.0009,E2 360.5506} C_DIS
LIN {X 5.4102,Y 113.8908,Z 117,A 82.4248,B 24.9343,C -1.8727,E1 25.009,E2 363.4633} C_DIS
LIN {X 11.2733,Y 113.461,Z 117,A 79.4254,B 24.9344,C -1.8706,E1 25.0173,E2 366.4662} C_DIS
LIN {X 15.9026,Y 112.9037,Z 117,A 77.1243,B 24.9344,C -1.8719,E1 25.0237,E2 368.7624} C_DIS
LIN {X 19.4465,Y 112.3494,Z 117,A 75.144,B 24.9349,C -1.8636,E1 25.0292,E2 370.7602} C_DIS
LIN {X 23.0695,Y 111.6599,Z 117,A 73.5441,B 24.9342,C -1.8737,E1 25.0335,E2 372.3342} C_DIS
LIN {X 25.8475,Y 111.0498,Z 117,A 72.0506,B 24.9344,C -1.8702,E1 25.0376,E2 373.8342} C_DIS
LIN {X 29.595,Y 110.1103,Z 117,A 70.0977,B 24.9346,C -1.8685,E1 25.0429,E2 375.7881} C_DIS
LIN {X 33.1976,Y 109.0798,Z 117,A 68.1057,B 24.935,C -1.8624,E1 25.0482,E2 377.7911} C_DIS
LIN {X 37.004,Y 107.848,Z 117,A 66.0253,B 24.9353,C -1.8576,E1 25.0538,E2 379.8787} C_DIS
LIN {X 40.9698,Y 106.4048,Z 117,A 63.8851,B 24.9355,C -1.8548,E1 25.0594,E2 382.0211} C_DIS
LIN {X 44.8633,Y 104.8228,Z 117,A 61.723,B 24.9358,C -1.8503,E1 25.0649,E2 384.1886} C_DIS
LIN {X 51.4409,Y 101.7556,Z 117,A 58.2799,B 24.9355,C -1.8548,E1 25.0736,E2 387.6122} C_DIS
LIN {X 54.9985,Y 99.8787,Z 117,A 55.8047,B 24.9371,C -1.8321,E1 25.0798,E2 390.1339} C_DIS
LIN {X 58.4708,Y 97.8855,Z 117,A 54.2321,B 24.936,C -1.8484,E1 25.0834,E2 391.6632} C_DIS
LIN {X 61.6598,Y 95.9073,Z 117,A 52.2078,B 24.9366,C -1.8393,E1 25.0882,E2 393.7023} C_DIS
LIN {X 65.4154,Y 93.3869,Z 117,A 50.242,B 24.9359,C -1.8491,E1 25.0927,E2 395.6383} C_DIS
LIN {X 68.3307,Y 91.2747,Z 117,A 48.3694,B 24.9363,C -1.8431,E1 25.0969,E2 397.5184} C_DIS
LIN {X 70.9522,Y 89.2525,Z 117,A 46.7392,B 24.9364,C -1.8415,E1 25.1005,E2 399.1464} C_DIS
LIN {X 74.2228,Y 86.5519,Z 117,A 44.3746,B 24.9374,C -1.827,E1 25.1056,E2 401.5362} C_DIS
LIN {X 79.4546,Y 81.7759,Z 117,A 41.005,B 24.9374,C -1.8281,E1 25.1125,E2 404.8893} C_DIS
LIN {X 82.2091,Y 79.0052,Z 117,A 38.7337,B 24.9386,C -1.81,E1 25.117,E2 407.1936} C_DIS
LIN {X 84.527,Y 76.5212,Z 117,A 37.5337,B 24.9373,C -1.829,E1 25.1191,E2 408.3436} C_DIS
LIN {X 86.1504,Y 74.6888,Z 117,A 36.0123,B 24.9384,C -1.813,E1 25.122,E2 409.8959} C_DIS
LIN {X 90.4664,Y 69.3976,Z 117,A 32.9523,B 24.9378,C -1.8215,E1 25.1273,E2 412.9215} C_DIS
LIN {X 91.9723,Y 67.3885,Z 117,A 31.5527,B 24.9385,C -1.8121,E1 25.1296,E2 414.3366} C_DIS
LIN {X 93.8128,Y 64.8028,Z 117,A 29.8163,B 24.9392,C -1.8016,E1 25.1324,E2 416.0893} C_DIS
LIN {X 96.0686,Y 61.4085,Z 117,A 28.1658,B 24.9383,C -1.8144,E1 25.1349,E2 417.7014} C_DIS
LIN {X 97.3517,Y 59.3532,Z 117,A 26.6989,B 24.9393,C -1.7998,E1 25.1371,E2 419.1954} C_DIS
LIN {X 99.03,Y 56.5094,Z 117,A 25.0415,B 24.9396,C -1.7953,E1 25.1394,E2 420.8546} C_DIS
LIN {X 100.7185,Y 53.4419,Z 117,A 23.2347,B 24.9401,C -1.7883,E1 25.1418,E2 422.6685} C_DIS
LIN {X 102.3617,Y 50.2237,Z 117,A 20.7056,B 24.9426,C -1.7508,E1 25.1451,E2 425.2725} C_DIS
LIN {X 104.4909,Y 45.6264,Z 117,A 19.3028,B 24.9396,C -1.7956,E1 25.1465,E2 426.5621} C_DIS
LIN {X 106.9535,Y 39.5131,Z 117,A 15.8283,B 24.9407,C -1.7783,E1 25.1502,E2 430.0582} C_DIS
LIN {X 107.7961,Y 37.1554,Z 117,A 14.4118,B 24.9415,C -1.7672,E1 25.1515,E2 431.4929} C_DIS
LIN {X 108.9444,Y 33.6343,Z 117,A 12.6131,B 24.9416,C -1.7645,E1 25.153,E2 433.2878} C_DIS
LIN {X 109.8395,Y 30.5888,Z 117,A 10.9912,B 24.9421,C -1.7583,E1 25.1542,E2 434.9149} C_DIS
LIN {X 110.7346,Y 27.1661,Z 117,A 9.2264,B 24.9424,C -1.7534,E1 25.1555,E2 436.6811} C_DIS
LIN {X 112.35,Y 19.4377,Z 117,A 5.1931,B 24.9434,C -1.7378,E1 25.1577,E2 440.7276} C_DIS
LIN {X 112.7903,Y 16.7008,Z 117,A 3.6326,B 24.9442,C -1.7257,E1 25.1583,E2 442.3076} C_DIS
LIN {X 113.5258,Y 10.5843,Z 117,A 0.9526,B 24.9436,C -1.735,E1 25.1592,E2 444.9499} C_DIS
LIN {X 113.8942,Y 5.3326,Z 117,A -1.8936,B 24.9447,C -1.7171,E1 25.1597,E2 447.8214} C_DIS
LIN {X 114.011,Y 1.4328,Z 117,A -4.1141,B 24.9459,C -1.6987,E1 25.1597,E2 450.072} C_DIS
LIN {X 113.8713,Y -5.8037,Z 117,A -7.3995,B 24.9456,C -1.7031,E1 25.1595,E2 453.3274} C_DIS
LIN {X 113.6541,Y -9.1037,Z 117,A -9.7029,B 24.9479,C -1.6681,E1 25.159,E2 455.6996} C_DIS
LIN {X 113.1794,Y -13.8154,Z 117,A -11.3278,B 24.9461,C -1.6952,E1 25.1585,E2 457.2512} C_DIS
LIN {X 112.1532,Y -20.5405,Z 117,A -14.6357,B 24.9465,C -1.6892,E1 25.1571,E2 460.5537} C_DIS
LIN {X 110.8239,Y -26.8,Z 117,A -18.0821,B 24.9479,C -1.668,E1 25.155,E2 464.03} C_DIS
LIN {X 109.7839,Y -30.7848,Z 117,A -20.0691,B 24.948,C -1.6652,E1 25.1535,E2 466.0122} C_DIS
LIN {X 108.0822,Y -36.3096,Z 117,A -22.6063,B 24.9475,C -1.6731,E1 25.1515,E2 468.5164} C_DIS
LIN {X 107.2465,Y -38.7098,Z 117,A -24.206,B 24.9487,C -1.6541,E1 25.1499,E2 470.1519} C_DIS
LIN {X 106.0877,Y -41.7795,Z 117,A -25.8025,B 24.9489,C -1.6514,E1 25.1483,E2 471.7459} C_DIS
LIN {X 104.8053,Y -44.9038,Z 117,A -27.5534,B 24.9494,C -1.6436,E1 25.1464,E2 473.5056} C_DIS
LIN {X 103.3938,Y -48.0608,Z 117,A -29.2249,B 24.9495,C -1.6414,E1 25.1445,E2 475.1732} C_DIS
LIN {X 101.8456,Y -51.2648,Z 117,A -32.1087,B 24.9529,C -1.5858,E1 25.1408,E2 478.1727} C_DIS
LIN {X 98.7894,Y -56.9279,Z 117,A -34.0564,B 24.9499,C -1.6352,E1 25.1383,E2 479.9938} C_DIS
LIN {X 97.4356,Y -59.2151,Z 117,A -35.5749,B 24.9507,C -1.6228,E1 25.136,E2 481.5337} C_DIS
LIN {X 94.0896,Y -64.4019,Z 117,A -38.8287,B 24.9516,C -1.607,E1 25.131,E2 484.8086} C_DIS
LIN {X 91.879,Y -67.5161,Z 117,A -40.538,B 24.9514,C -1.6113,E1 25.1282,E2 486.4995} C_DIS
LIN {X 90.2193,Y -69.7182,Z 117,A -41.9143,B 24.9516,C -1.608,E1 25.1259,E2 487.8771} C_DIS
LIN {X 87.2461,Y -73.4078,Z 117,A -44.281,B 24.9519,C -1.6023,E1 25.1217,E2 490.2464} C_DIS
LIN {X 83.5123,Y -77.629,Z 117,A -47.2476,B 24.9527,C -1.5888,E1 25.1161,E2 493.2316} C_DIS
LIN {X 79.4774,Y -81.754,Z 117,A -49.9286,B 24.9525,C -1.5916,E1 25.1109,E2 495.8945} C_DIS
LIN {X 75.5402,Y -85.4065,Z 117,A -52.6088,B 24.9529,C -1.5861,E1 25.1054,E2 498.577} C_DIS
LIN {X 70.234,Y -89.8201,Z 117,A -57.0945,B 24.956,C -1.5325,E1 25.0954,E2 503.1723} C_DIS
LIN {X 65.485,Y -93.3385,Z 117,A -58.9295,B 24.9534,C -1.5773,E1 25.0915,E2 504.8949} C_DIS
LIN {X 63.1853,Y -94.9105,Z 117,A -60.3867,B 24.9537,C -1.5719,E1 25.0881,E2 506.36} C_DIS
LIN {X 60.5828,Y -96.5914,Z 117,A -62.3897,B 24.9551,C -1.5488,E1 25.0833,E2 508.4111} C_DIS
LIN {X 57.7899,Y -98.2879,Z 117,A -63.8419,B 24.9547,C -1.5543,E1 25.0798,E2 509.846} C_DIS
LIN {X 54.7114,Y -100.0347,Z 117,A -65.4859,B 24.9546,C -1.5571,E1 25.0758,E2 511.4784} C_DIS
LIN {X 51.9296,Y -101.5059,Z 117,A -67.0018,B 24.9546,C -1.5574,E1 25.0721,E2 512.9894} C_DIS
LIN {X 47.4843,Y -103.6622,Z 117,A -69.5876,B 24.9551,C -1.5488,E1 25.0655,E2 515.589} C_DIS
LIN {X 43.1882,Y -105.5223,Z 117,A -71.9344,B 24.9552,C -1.5456,E1 25.0595,E2 517.9378} C_DIS
LIN {X 40.1782,Y -106.7046,Z 117,A -73.4385,B 24.9551,C -1.5487,E1 25.0556,E2 519.4312} C_DIS
LIN {X 36.7963,Y -107.9181,Z 117,A -75.2829,B 24.9553,C -1.5446,E1 25.0507,E2 521.2815} C_DIS
LIN {X 33.5035,Y -108.9849,Z 117,A -76.9719,B 24.9553,C -1.5448,E1 25.0462,E2 522.967} C_DIS
LIN {X 30.2709,Y -109.9277,Z 117,A -78.7831,B 24.9557,C -1.5376,E1 25.0413,E2 524.7922} C_DIS
LIN {X 26.7475,Y -110.8367,Z 117,A -80.4623,B 24.9554,C -1.5424,E1 25.0368,E2 526.4577} C_DIS
LIN {X 21.3903,Y -111.9938,Z 117,A -83.7681,B 24.957,C -1.5158,E1 25.0276,E2 529.8224} C_DIS
LIN {X 17.5033,Y -112.6666,Z 117,A -85.1639,B 24.9556,C -1.5399,E1 25.0239,E2 531.1596} C_DIS
LIN {X 14.4354,Y -113.1008,Z 117,A -87.6405,B 24.9579,C -1.4989,E1 25.0168,E2 533.7313} C_DIS
LIN {X 9.0388,Y -113.6593,Z 117,A -89.3739,B 24.9555,C -1.5406,E1 25.0123,E2 535.3651} C_DIS
LIN {X 3.0945,Y -113.9768,Z 117,A -92.4274,B 24.9558,C -1.5366,E1 25.0037,E2 538.4269} C_DIS
LIN {X 0.8022,Y -114.0135,Z 117,A -93.1716,B 24.9547,C -1.5542,E1 25.0017,E2 539.1295} C_DIS
Enddeposition()
LIN {X 0.8022,Y -114.0135,Z 117,A -93.1716,B 24.9547,C -1.5542,E1 25.0017,E2 539.1295} C_DIS
Startdeposition()
$VEL.CP = VEL_PRINT
LIN {X 2.5805,Y -113.0877,Z 117,A -92.1574,B 24.9535,C -1.575,E1 25.0047,E2 538.066} C_DIS
LIN {X 9.2421,Y -112.7381,Z 117,A -89.1258,B 24.9543,C -1.5612,E1 25.0131,E2 535.0683} C_DIS
LIN {X 15.3239,Y -112.0748,Z 117,A -85.5369,B 24.953,C -1.5843,E1 25.0232,E2 531.427} C_DIS
LIN {X 24.5909,Y -110.4118,Z 117,A -80.7796,B 24.9528,C -1.5876,E1 25.0363,E2 526.6674} C_DIS
LIN {X 28.0657,Y -109.579,Z 117,A -78.9378,B 24.9526,C -1.5909,E1 25.0412,E2 524.8205} C_DIS
LIN {X 31.5162,Y -108.639,Z 117,A -77.2362,B 24.9528,C -1.588,E1 25.0458,E2 523.1287} C_DIS
LIN {X 34.082,Y -107.8612,Z 117,A -75.7472,B 24.9523,C -1.5954,E1 25.0498,E2 521.6248} C_DIS
LIN {X 37.5538,Y -106.7004,Z 117,A -73.9539,B 24.9523,C -1.5951,E1 25.0545,E2 519.8357} C_DIS
LIN {X 41.9193,Y -105.0637,Z 117,A -71.1487,B 24.9509,C -1.6184,E1 25.0619,E2 516.9817} C_DIS
LIN {X 45.2187,Y -103.6847,Z 117,A -69.7904,B 24.952,C -1.6006,E1 25.0653,E2 515.6686} C_DIS
LIN {X 48.3765,Y -102.2518,Z 117,A -67.0361,B 24.9491,C -1.6488,E1 25.0726,E2 512.8076} C_DIS
LIN {X 53.7667,Y -99.521,Z 117,A -65.2972,B 24.9524,C -1.5939,E1 25.0765,E2 511.2033} C_DIS
LIN {X 59.9953,Y -95.8948,Z 117,A -61.0958,B 24.9505,C -1.6256,E1 25.0867,E2 506.94} C_DIS
LIN {X 63.1286,Y -93.8623,Z 117,A -59.3904,B 24.9508,C -1.6208,E1 25.0907,E2 505.2515} C_DIS
LIN {X 68.4182,Y -90.0791,Z 117,A -56.3178,B 24.951,C -1.6176,E1 25.0976,E2 502.1973} C_DIS
LIN {X 70.4385,Y -88.5088,Z 117,A -54.5019,B 24.9493,C -1.6443,E1 25.1017,E2 500.3252} C_DIS
LIN {X 73.1069,Y -86.3176,Z 117,A -53.4021,B 24.9509,C -1.6185,E1 25.1039,E2 499.2905} C_DIS
LIN {X 74.8518,Y -84.8103,Z 117,A -51.4532,B 24.9485,C -1.6571,E1 25.1081,E2 497.2584} C_DIS
LIN {X 77.8622,Y -82.0547,Z 117,A -50.0377,B 24.9501,C -1.632,E1 25.1109,E2 495.9079} C_DIS
LIN {X 81.5268,Y -78.4133,Z 117,A -47.339,B 24.9495,C -1.6422,E1 25.1162,E2 493.1965} C_DIS
LIN {X 85.3893,Y -74.1889,Z 117,A -44.5258,B 24.9493,C -1.6456,E1 25.1215,E2 490.3876} C_DIS
LIN {X 87.536,Y -71.6443,Z 117,A -42.665,B 24.9485,C -1.6582,E1 25.1248,E2 488.5059} C_DIS
LIN {X 89.6587,Y -68.9678,Z 117,A -41.1458,B 24.9488,C -1.6531,E1 25.1274,E2 487.0058} C_DIS
LIN {X 91.4732,Y -66.5433,Z 117,A -39.1705,B 24.9472,C -1.6778,E1 25.1307,E2 484.9817} C_DIS
LIN {X 93.396,Y -63.8173,Z 117,A -37.1024,B 24.9458,C -1.7002,E1 25.134,E2 482.8709} C_DIS
LIN {X 96.1161,Y -59.641,Z 117,A -35.466,B 24.948,C -1.6661,E1 25.1363,E2 481.3234} C_DIS
LIN {X 99.0036,Y -54.7119,Z 117,A -31.9292,B 24.9456,C -1.7045,E1 25.1413,E2 477.7142} C_DIS
LIN {X 100.9564,Y -51.0225,Z 117,A -30.4761,B 24.9471,C -1.68,E1 25.1431,E2 476.3267} C_DIS
LIN {X 102.2283,Y -48.4254,Z 117,A -28.8529,B 24.9464,C -1.6918,E1 25.1451,E2 474.6845} C_DIS
LIN {X 104.0862,Y -44.2884,Z 117,A -26.607,B 24.9461,C -1.6964,E1 25.1476,E2 472.4398} C_DIS
LIN {X 105.3425,Y -41.2095,Z 117,A -25.0093,B 24.946,C -1.6977,E1 25.1492,E2 470.848} C_DIS
LIN {X 106.6088,Y -37.8146,Z 117,A -22.17,B 24.9426,C -1.7505,E1 25.152,E2 467.8999} C_DIS
LIN {X 108.4396,Y -32.1882,Z 117,A -20.2261,B 24.9452,C -1.7106,E1 25.1535,E2 466.0614} C_DIS
LIN {X 109.2302,Y -29.394,Z 117,A -18.7148,B 24.9447,C -1.7171,E1 25.1546,E2 464.5433} C_DIS
LIN {X 111.0218,Y -21.6675,Z 117,A -14.9653,B 24.9447,C -1.7175,E1 25.157,E2 460.8146} C_DIS
LIN {X 112.2167,Y -14.2383,Z 117,A -11.4466,B 24.9448,C -1.7162,E1 25.1585,E2 457.3197} C_DIS
LIN {X 112.8434,Y -7.8524,Z 117,A -7.6421,B 24.9424,C -1.7524,E1 25.1595,E2 453.4523} C_DIS
LIN {X 113.1012,Y -1.8491,Z 117,A -4.0094,B 24.9399,C -1.79,E1 25.1598,E2 449.7527} C_DIS
LIN {X 113.0824,Y 2.8302,Z 117,A -2.4085,B 24.9418,C -1.7616,E1 25.1598,E2 448.2282} C_DIS
LIN {X 112.7799,Y 8.7193,Z 117,A 0.6178,B 24.9411,C -1.7731,E1 25.1592,E2 445.1928} C_DIS
LIN {X 112.0937,Y 15.1869,Z 117,A 3.832,B 24.9406,C -1.7799,E1 25.1582,E2 441.9817} C_DIS
LIN {X 111.5368,Y 18.8367,Z 117,A 6.7452,B 24.9369,C -1.8346,E1 25.1568,E2 438.9564} C_DIS
LIN {X 110.3831,Y 24.7228,Z 117,A 8.7091,B 24.9397,C -1.7939,E1 25.1557,E2 437.1001} C_DIS
LIN {X 109.5212,Y 28.2908,Z 117,A 10.6531,B 24.939,C -1.8036,E1 25.1544,E2 435.1444} C_DIS
LIN {X 108.442,Y 32.1802,Z 117,A 12.6323,B 24.9388,C -1.8068,E1 25.1529,E2 433.1689} C_DIS
LIN {X 107.4787,Y 35.2674,Z 117,A 14.235,B 24.9386,C -1.8102,E1 25.1515,E2 431.5674} C_DIS
LIN {X 106.6016,Y 37.8352,Z 117,A 15.5924,B 24.9384,C -1.8135,E1 25.1503,E2 430.2097} C_DIS
LIN {X 104.4822,Y 43.3477,Z 117,A 18.7013,B 24.9374,C -1.8277,E1 25.1471,E2 427.0846} C_DIS
LIN {X 101.6382,Y 49.6522,Z 117,A 22.0342,B 24.9372,C -1.8298,E1 25.1432,E2 423.7646} C_DIS
LIN {X 99.7613,Y 53.3235,Z 117,A 24.1771,B 24.9367,C -1.8382,E1 25.1404,E2 421.6136} C_DIS
LIN {X 97.437,Y 57.4568,Z 117,A 26.5609,B 24.9363,C -1.8439,E1 25.1371,E2 419.2285} C_DIS
LIN {X 95.8256,Y 60.106,Z 117,A 28.1178,B 24.936,C -1.8474,E1 25.1348,E2 417.6711} C_DIS
LIN {X 93.7458,Y 63.3008,Z 117,A 29.7652,B 24.9366,C -1.8395,E1 25.1324,E2 416.0506} C_DIS
LIN {X 92.5459,Y 65.045,Z 117,A 31.1435,B 24.9354,C -1.8562,E1 25.1301,E2 414.6398} C_DIS
LIN {X 90.523,Y 67.8295,Z 117,A 32.8297,B 24.9353,C -1.8579,E1 25.1273,E2 412.9576} C_DIS
LIN {X 86.7017,Y 72.6517,Z 117,A 35.7781,B 24.9353,C -1.8578,E1 25.1222,E2 410.0233} C_DIS
LIN {X 83.9194,Y 75.849,Z 117,A 38.5828,B 24.9329,C -1.8926,E1 25.1169,E2 407.1489} C_DIS
LIN {X 81.3931,Y 78.5519,Z 117,A 39.918,B 24.9343,C -1.8723,E1 25.1144,E2 405.8675} C_DIS
LIN {X 79.6152,Y 80.3536,Z 117,A 41.4075,B 24.9334,C -1.8844,E1 25.1114,E2 404.3557} C_DIS
LIN {X 74.1197,Y 85.4498,Z 117,A 44.9137,B 24.9338,C -1.879,E1 25.1042,E2 400.8763} C_DIS
LIN {X 71.9591,Y 87.2773,Z 117,A 46.6314,B 24.9327,C -1.8945,E1 25.1005,E2 399.1285} C_DIS
LIN {X 69.0591,Y 89.5884,Z 117,A 48.3289,B 24.933,C -1.8899,E1 25.0968,E2 397.4483} C_DIS
LIN {X 66.2866,Y 91.6612,Z 117,A 50.1564,B 24.9326,C -1.8963,E1 25.0926,E2 395.6122} C_DIS
LIN {X 63.4273,Y 93.6601,Z 117,A 52.3037,B 24.9312,C -1.9163,E1 25.0876,E2 393.4248} C_DIS
LIN {X 60.2601,Y 95.7294,Z 117,A 53.7597,B 24.9324,C -1.8987,E1 25.0843,E2 392.0152} C_DIS
LIN {X 54.1521,Y 99.3119,Z 117,A 57.0462,B 24.933,C -1.8906,E1 25.0764,E2 388.7578} C_DIS
LIN {X 51.5514,Y 100.6861,Z 117,A 58.7689,B 24.9321,C -1.9028,E1 25.0721,E2 387.0109} C_DIS
LIN {X 45.8423,Y 103.4127,Z 117,A 61.9315,B 24.932,C -1.9047,E1 25.0641,E2 383.8519} C_DIS
LIN {X 43.1941,Y 104.546,Z 117,A 63.5864,B 24.9313,C -1.9149,E1 25.0598,E2 382.1768} C_DIS
LIN {X 40.326,Y 105.6841,Z 117,A 64.883,B 24.932,C -1.9048,E1 25.0565,E2 380.9069} C_DIS
LIN {X 36.2041,Y 107.1658,Z 117,A 66.967,B 24.9323,C -1.9009,E1 25.051,E2 378.8364} C_DIS
LIN {X 33.8199,Y 107.9424,Z 117,A 68.5166,B 24.9313,C -1.9141,E1 25.0468,E2 377.2585} C_DIS
LIN {X 30.6258,Y 108.8915,Z 117,A 70.2332,B 24.9311,C -1.9165,E1 25.0422,E2 375.539} C_DIS
LIN {X 26.8761,Y 109.8768,Z 117,A 72.1744,B 24.9311,C -1.9168,E1 25.037,E2 373.6002} C_DIS
LIN {X 22.6117,Y 110.8331,Z 117,A 74.5282,B 24.9306,C -1.9239,E1 25.0305,E2 371.2325} C_DIS
LIN {X 18.5927,Y 111.5776,Z 117,A 76.4346,B 24.9311,C -1.9176,E1 25.0253,E2 369.3431} C_DIS
LIN {X 14.7405,Y 112.1517,Z 117,A 78.7557,B 24.9299,C -1.9331,E1 25.0188,E2 366.9872} C_DIS
LIN {X 11.5098,Y 112.5293,Z 117,A 79.8614,B 24.9316,C -1.9101,E1 25.0159,E2 365.9368} C_DIS
LIN {X 5.998,Y 112.9572,Z 117,A 82.9255,B 24.9308,C -1.9214,E1 25.0073,E2 362.8474} C_DIS
LIN {X -1.1273,Y 113.1113,Z 117,A 87.0014,B 24.9294,C -1.9406,E1 24.9958,E2 358.7261} C_DIS
LIN {X -5.1533,Y 112.999,Z 117,A 88.4199,B 24.9314,C -1.9135,E1 24.992,E2 357.3716} C_DIS
LIN {X -8.2549,Y 112.8162,Z 117,A 90.6873,B 24.9293,C -1.9423,E1 24.9855,E2 355.0352} C_DIS
LIN {X -12.5764,Y 112.4163,Z 117,A 92.1559,B 24.9316,C -1.9102,E1 24.9816,E2 353.6418} C_DIS
LIN {X -17.2053,Y 111.7999,Z 117,A 94.2917,B 24.9324,C -1.8991,E1 24.9758,E2 351.5307} C_DIS
LIN {X -21.312,Y 111.0903,Z 117,A 97.0325,B 24.9306,C -1.9238,E1 24.9681,E2 348.7284} C_DIS
LIN {X -25.4227,Y 110.2222,Z 117,A 98.868,B 24.9316,C -1.9097,E1 24.9631,E2 346.9243} C_DIS
LIN {X -28.5554,Y 109.4532,Z 117,A 100.6389,B 24.9313,C -1.9137,E1 24.9583,E2 345.1411} C_DIS
LIN {X -34.6269,Y 107.6859,Z 117,A 104.2544,B 24.9304,C -1.9273,E1 24.9486,E2 341.4871} C_DIS
LIN {X -38.3705,Y 106.4101,Z 117,A 106.3541,B 24.9303,C -1.9287,E1 24.943,E2 339.3798} C_DIS
LIN {X -42.3817,Y 104.8767,Z 117,A 108.3717,B 24.931,C -1.9191,E1 24.9378,E2 337.3806} C_DIS
LIN {X -45.778,Y 103.4408,Z 117,A 109.6856,B 24.9328,C -1.8935,E1 24.9346,E2 336.1245} C_DIS
LIN {X -49.5543,Y 101.6858,Z 117,A 112.789,B 24.9301,C -1.9312,E1 24.9266,E2 332.9235} C_DIS
LIN {X -54.3749,Y 99.191,Z 117,A 114.4728,B 24.9336,C -1.8826,E1 24.9227,E2 331.3504} C_DIS
LIN {X -57.71,Y 97.2873,Z 117,A 116.603,B 24.9333,C -1.8867,E1 24.9175,E2 329.2043} C_DIS
LIN {X -61.8648,Y 94.7007,Z 117,A 119.9082,B 24.9312,C -1.9157,E1 24.9096,E2 325.8193} C_DIS
LIN {X -66.0587,Y 91.8242,Z 117,A 122.0576,B 24.9328,C -1.893,E1 24.9048,E2 323.7167} C_DIS
LIN {X -68.6414,Y 89.9103,Z 117,A 123.5564,B 24.9334,C -1.8842,E1 24.9015,E2 322.2332} C_DIS
LIN {X -73.9416,Y 85.6053,Z 117,A 126.7174,B 24.9348,C -1.8645,E1 24.8948,E2 319.1071} C_DIS
LIN {X -76.1924,Y 83.6069,Z 117,A 128.9557,B 24.933,C -1.8898,E1 24.89,E2 316.7996} C_DIS
LIN {X -79.2985,Y 80.6663,Z 117,A 131.1952,B 24.9332,C -1.8875,E1 24.8855,E2 314.556} C_DIS
LIN {X -82.4761,Y 77.4141,Z 117,A 132.4055,B 24.9367,C -1.8379,E1 24.8834,E2 313.4588} C_DIS
LIN {X -87.1779,Y 72.0787,Z 117,A 136.3464,B 24.9364,C -1.842,E1 24.8761,E2 309.4903} C_DIS
LIN {X -90.4889,Y 67.875,Z 117,A 139.1899,B 24.9365,C -1.84,E1 24.8712,E2 306.6381} C_DIS
LIN {X -93.5895,Y 63.5316,Z 117,A 142.4935,B 24.9354,C -1.8565,E1 24.8659,E2 303.2789} C_DIS
LIN {X -95.8747,Y 60.0274,Z 117,A 144.0434,B 24.9374,C -1.8277,E1 24.8637,E2 301.7898} C_DIS
LIN {X -97.632,Y 57.1269,Z 117,A 145.7032,B 24.9379,C -1.8204,E1 24.8613,E2 300.1388} C_DIS
LIN {X -99.086,Y 54.5679,Z 117,A 147.4028,B 24.9376,C -1.8243,E1 24.859,E2 298.421} C_DIS
LIN {X -100.752,Y 51.4226,Z 117,A 149.0801,B 24.9383,C -1.814,E1 24.8568,E2 296.7594} C_DIS
LIN {X -103.6571,Y 45.2819,Z 117,A 152.5147,B 24.939,C -1.8033,E1 24.8528,E2 293.3315} C_DIS
LIN {X -104.8287,Y 42.4996,Z 117,A 154.0419,B 24.9394,C -1.7985,E1 24.8512,E2 291.8072} C_DIS
LIN {X -105.8806,Y 39.8071,Z 117,A 155.5226,B 24.9396,C -1.7946,E1 24.8497,E2 290.3275} C_DIS
LIN {X -107.1356,Y 36.2936,Z 117,A 157.4806,B 24.9399,C -1.7914,E1 24.8479,E2 288.3661} C_DIS
LIN {X -107.9068,Y 33.9347,Z 117,A 158.6948,B 24.9402,C -1.7857,E1 24.8469,E2 287.1585} C_DIS
LIN {X -108.9267,Y 30.5015,Z 117,A 160.6781,B 24.9402,C -1.7866,E1 24.8453,E2 285.1615} C_DIS
LIN {X -109.8523,Y 26.9765,Z 117,A 162.393,B 24.9409,C -1.7756,E1 24.8442,E2 283.463} C_DIS
LIN {X -110.5586,Y 23.9181,Z 117,A 164.0025,B 24.9412,C -1.7712,E1 24.8432,E2 281.8544} C_DIS
LIN {X -111.2943,Y 20.2202,Z 117,A 165.9198,B 24.9416,C -1.7653,E1 24.8422,E2 279.9397} C_DIS
LIN {X -111.8451,Y 16.9129,Z 117,A 167.6165,B 24.942,C -1.7598,E1 24.8414,E2 278.2463} C_DIS
LIN {X -112.3342,Y 13.2774,Z 117,A 169.5102,B 24.9423,C -1.7552,E1 24.8408,E2 276.3522} C_DIS
LIN {X -112.688,Y 9.8464,Z 117,A 171.2169,B 24.9427,C -1.7479,E1 24.8403,E2 274.6527} C_DIS
LIN {X -112.9231,Y 6.615,Z 117,A 172.9606,B 24.9428,C -1.7466,E1 24.84,E2 272.9015} C_DIS
LIN {X -113.1155,Y -0.2906,Z 117,A 176.2107,B 24.9442,C -1.7253,E1 24.8398,E2 269.6825} C_DIS
LIN {X -113.0457,Y -4.0277,Z 117,A 178.6375,B 24.9432,C -1.7403,E1 24.84,E2 267.2055} C_DIS
LIN {X -112.7571,Y -9.0038,Z 117,A -179.0642,B 24.9444,C -1.7231,E1 24.8404,E2 264.9342} C_DIS
LIN {X -112.3893,Y -12.8066,Z 117,A -177.1406,B 24.9448,C -1.7165,E1 24.841,E2 263.015} C_DIS
LIN {X -111.994,Y -15.893,Z 117,A -175.5758,B 24.9451,C -1.711,E1 24.8416,E2 261.4538} C_DIS
LIN {X -111.4301,Y -19.4653,Z 117,A -173.6588,B 24.9453,C -1.7086,E1 24.8424,E2 259.5314} C_DIS
LIN {X -110.8336,Y -22.6089,Z 117,A -172.0707,B 24.9457,C -1.7022,E1 24.8433,E2 257.9491} C_DIS
LIN {X -110.0662,Y -26.0978,Z 117,A -170.0047,B 24.9454,C -1.7067,E1 24.8446,E2 255.8601} C_DIS
LIN {X -108.8782,Y -30.6726,Z 117,A -167.8,B 24.9464,C -1.6918,E1 24.8462,E2 253.6781} C_DIS
LIN {X -107.0474,Y -36.5551,Z 117,A -165.0326,B 24.9478,C -1.6683,E1 24.8485,E2 250.9508} C_DIS
LIN {X -105.6578,Y -40.3955,Z 117,A -162.5729,B 24.9473,C -1.6777,E1 24.8509,E2 248.4549} C_DIS
LIN {X -104.1434,Y -44.1526,Z 117,A -160.5062,B 24.9476,C -1.6723,E1 24.8531,E2 246.3896} C_DIS
LIN {X -102.5581,Y -47.7188,Z 117,A -158.5915,B 24.9481,C -1.6641,E1 24.8553,E2 244.4839} C_DIS
LIN {X -100.9689,Y -50.9981,Z 117,A -155.5813,B 24.9454,C -1.7061,E1 24.8593,E2 241.3574} C_DIS
LIN {X -97.8505,Y -56.7514,Z 117,A -153.7495,B 24.9498,C -1.637,E1 24.8616,E2 239.6807} C_DIS
LIN {X -94.5557,Y -62.0847,Z 117,A -150.3386,B 24.9498,C -1.638,E1 24.8666,E2 236.25} C_DIS
LIN {X -92.639,Y -64.911,Z 117,A -148.4955,B 24.9498,C -1.6381,E1 24.8695,E2 234.3975} C_DIS
LIN {X -90.8315,Y -67.4189,Z 117,A -146.7387,B 24.9495,C -1.642,E1 24.8725,E2 232.6231} C_DIS
LIN {X -88.7218,Y -70.1689,Z 117,A -145.116,B 24.9501,C -1.6323,E1 24.8752,E2 231.0157} C_DIS
LIN {X -86.3323,Y -73.0896,Z 117,A -143.1535,B 24.9502,C -1.6299,E1 24.8787,E2 229.0498} C_DIS
LIN {X -82.0159,Y -77.9034,Z 117,A -139.918,B 24.9508,C -1.6209,E1 24.8848,E2 225.8216} C_DIS
LIN {X -77.0701,Y -82.7996,Z 117,A -136.3491,B 24.9511,C -1.6152,E1 24.892,E2 222.2513} C_DIS
LIN {X -74.4422,Y -85.1681,Z 117,A -134.5459,B 24.9513,C -1.6121,E1 24.8957,E2 220.4483} C_DIS
LIN {X -71.7001,Y -87.4912,Z 117,A -132.7048,B 24.9515,C -1.6094,E1 24.8997,E2 218.6064} C_DIS
LIN {X -68.9427,Y -89.6781,Z 117,A -130.9243,B 24.9517,C -1.6061,E1 24.9036,E2 216.8273} C_DIS
LIN {X -65.8904,Y -91.9443,Z 117,A -128.3657,B 24.9503,C -1.6292,E1 24.9095,E2 214.2049} C_DIS
LIN {X -62.2621,Y -94.4387,Z 117,A -127.1474,B 24.953,C -1.5834,E1 24.9121,E2 213.0914} C_DIS
LIN {X -58.8389,Y -96.6087,Z 117,A -124.7549,B 24.9524,C -1.5943,E1 24.9178,E2 210.6655} C_DIS
LIN {X -56.3913,Y -98.0575,Z 117,A -123.2548,B 24.9524,C -1.5947,E1 24.9215,E2 209.1599} C_DIS
LIN {X -53.3587,Y -99.7422,Z 117,A -120.8118,B 24.9508,C -1.6212,E1 24.9277,E2 206.647} C_DIS
LIN {X -49.296,Y -101.8099,Z 117,A -119.4058,B 24.9532,C -1.5803,E1 24.931,E2 205.3346} C_DIS
LIN {X -45.7886,Y -103.4362,Z 117,A -117.0583,B 24.9524,C -1.5944,E1 24.937,E2 202.9478} C_DIS
LIN {X -42.0592,Y -105.0079,Z 117,A -114.7575,B 24.9519,C -1.603,E1 24.943,E2 200.6216} C_DIS
LIN {X -38.9675,Y -106.1924,Z 117,A -113.7623,B 24.9537,C -1.5726,E1 24.9454,E2 199.6965} C_DIS
LIN {X -36.6544,Y -107.014,Z 117,A -112.2203,B 24.953,C -1.5841,E1 24.9496,E2 198.1241} C_DIS
LIN {X -33.6088,Y -108.0079,Z 117,A -110.6141,B 24.953,C -1.5822,E1 24.9539,E2 196.5196} C_DIS
LIN {X -30.384,Y -108.96,Z 117,A -108.9705,B 24.9533,C -1.5785,E1 24.9582,E2 194.8822} C_DIS
LIN {X -27.1342,Y -109.8139,Z 117,A -106.4213,B 24.9512,C -1.614,E1 24.9654,E2 192.2451} C_DIS
LIN {X -22.156,Y -110.9266,Z 117,A -104.496,B 24.953,C -1.5844,E1 24.9705,E2 190.3879} C_DIS
LIN {X -18.5196,Y -111.5898,Z 117,A -102.2655,B 24.9521,C -1.5993,E1 24.9767,E2 188.1198} C_DIS
LIN {X -14.8172,Y -112.1417,Z 117,A -101.0941,B 24.954,C -1.5675,E1 24.9798,E2 187.0228} C_DIS
LIN {X -9.1821,Y -112.7429,Z 117,A -98.2754,B 24.9541,C -1.5649,E1 24.9876,E2 184.2085} C_DIS
LIN {X -2.8983,Y -113.0804,Z 117,A -93.905,B 24.951,C -1.6169,E1 25.0001,E2 179.7142} C_DIS
LIN {X 0.8034,Y -113.0853,Z 117,A -93.7311,B 24.9554,C -1.5435,E1 25.0001,E2 179.7142} C_DIS
Enddeposition()
LIN {X 0.8034,Y -113.0853,Z 117,A -93.7311,B 24.9554,C -1.5435,E1 25.0001,E2 179.7142} C_DIS
Startdeposition()
$VEL.CP = VEL_PRINT
Enddeposition()
END
